(* IEC 61131-3 sources: std_i2980_v2.06_cp053/Source/IMM/ieccontrol/ODC1 (part 9) *)

END_TRANSITION
(* end sfc-code *)

END_ALGORITHM

(*
Run the auto cycle.
When the cycle has finished and mbStopCycle OR mbStopAfterCycle are true
opmode is automatically switched to manual and the PROCESS_ALGORITHM stops itself.
*)

PROCESS_ALGORITHM paRunAutomaticMovements ON TaskSequencer

#BEGIN_EDIT_BLOCK
(**************************************** WARNING ********************************************
 *** The KEBA Kemro K2 System including software is not intended for safety control tasks! ***
 ***                       For further information see Comment tab!                        ***
 *********************************************************************************************)

//call autoCycle
aRunAutoCycle(bStopCycle := mbStopCycle,
              bStopAfterCycle := mbStopAfterCycle);

IF aRunAutoCycle.bReady AND (mbStopCycle OR mbStopAfterCycle) THEN
   sv_bAutoCycleRunning := FALSE;
   // switch to manual mode and stop self at end of cycle
   fbAutoManual();

   abInterpreter.aResetStepMode();
   STOP_PROCESS_ALGORITHM(paCycleTime);
   STOP_PROCESS_ALGORITHM(paCycleTimeMachine);
   STOP_PROCESS_ALGORITHM();
END_IF;

;#END_EDIT_BLOCK END_ALGORITHM

(*
Cause initialisation of ODC sequence after startup(sv_bInitDone)
*)

POSTUPDATE_ALGORITHM pInitDone ON PU_Task_3 WITH sv_bInitDone

#BEGIN_EDIT_BLOCK
(**************************************** WARNING ********************************************
 *** The KEBA Kemro K2 System including software is not intended for safety control tasks! ***
 ***                       For further information see Comment tab!                        ***
 *********************************************************************************************)

fbDebugTrace2(nODCInterpreter,'Reloading ODC files because of sv_bInitDone');

IF sv_bUseProgramSwitches THEN
   //use program switches
   aSetPendingRecalc(RecalcMode := nODCRecalcReloadFiles);
ELSE
   //use existing sequence and only recalc internal arrays
   aSetPendingRecalc(RecalcMode := nODCRecalcInternal);
END_IF;

aDoPendingRecalc();
IF aDoPendingRecalc.bStartedRecalc THEN
   fbDebugTrace2(nDeviceState, 'recalc because pInitDone');
END_IF;

;#END_EDIT_BLOCK END_ALGORITHM

PROCESS_ALGORITHM paInit ON TaskMid AUTOSTART

VAR
 swoState : KSWO_Status;
END_VAR
#BEGIN_EDIT_BLOCK
(**************************************** WARNING ********************************************
 *** The KEBA Kemro K2 System including software is not intended for safety control tasks! ***
 ***                       For further information see Comment tab!                        ***
 *********************************************************************************************)

//initialize semaphore
Status := MovementsSema.Put();
IF Status <> KRTOS_Status_OK THEN
   dummy2 := ASSERT(FALSE, erAssert);
END_IF;

swoState := KSWO_AddVariable(Task := TaskInject,
                           Name := 'ActCycleTime',
                           Variable := sv_dCycleTime);

swoState := KSWO_AddVariable(Task := TaskAnalog,
                           Name := 'ActCycleTime',
                           Variable := sv_dCycleTime);

STOP_PROCESS_ALGORITHM();

;#END_EDIT_BLOCK END_ALGORITHM

(*
React to to operation mode changes and stop the autocycle immediately
when switching to setup/manual mode,
or reset cycle data when switching to Full/Halfauto operation mode.
*)

POSTUPDATE_ALGORITHM pOpmodeChanged ON PU_Task_7 WITH sv_OperationMode

#BEGIN_EDIT_BLOCK
(**************************************** WARNING ********************************************
 *** The KEBA Kemro K2 System including software is not intended for safety control tasks! ***
 ***                       For further information see Comment tab!                        ***
 *********************************************************************************************)

IF sv_OperationMode >= nHalfAutomatic THEN
   mbStopCycle := FALSE;
   mbStopAfterCycle := FALSE;
   (* back up sequence when machine is switched to auto mode
      and the sequence has changed *)
   START_PROCESS_ALGORITHM(paBackupSequence);

   (* PA stops itself again when finished *)
   START_PROCESS_ALGORITHM(paRunAutomaticMovements);
   START_PROCESS_ALGORITHM(paCycleTime);
   START_PROCESS_ALGORITHM(paCycleTimeMachine);
ELSIF sv_OperationMode < nHalfAutomatic THEN
   sv_bFirstCycle := TRUE;
   mbStopCycle := TRUE;
   mbCycleTimeRunning := FALSE;

   IF sv_StartedManualMovements.iStartedMovements = 0 THEN
      //recalc of sequence only if no movement is active
      //if there is still a movement active, the creation of a new sequence
      //will be triggered by postupdate algo pActiveMovements
      aDoPendingRecalc();
      IF aDoPendingRecalc.bStartedRecalc THEN
         fbDebugTrace2(nDeviceState, 'recalc because opmode change away from auto cycle');
      END_IF;
   END_IF;

END_IF;

;#END_EDIT_BLOCK END_ALGORITHM

(*
Handle evAlarmFinishCycleAndStop event which signals to stop after the end
of the current autocycle
*)

EVENT_ALGORITHM evaFinishCycleAndStop ON EV_Task_3 WITH evAlarmFinishCycleAndStop

VAR_INPUT
 evFinishCycleAndStopData : ALARM_EVENT_DATA;
END_VAR
#BEGIN_EDIT_BLOCK
(**************************************** WARNING ********************************************
 *** The KEBA Kemro K2 System including software is not intended for safety control tasks! ***
 ***                       For further information see Comment tab!                        ***
 *********************************************************************************************)

mbStopAfterCycle := TRUE;

;#END_EDIT_BLOCK END_ALGORITHM

POSTUPDATE_ALGORITHM pDataState ON PU_Task_3(1) WITH sv_DataState

VAR
 PrevState : tnDataState;
END_VAR
#BEGIN_EDIT_BLOCK
(**************************************** WARNING ********************************************
 *** The KEBA Kemro K2 System including software is not intended for safety control tasks! ***
 ***                       For further information see Comment tab!                        ***
 *********************************************************************************************)

IF sv_DataState = nReadMoldData THEN
   //loading of mold data in progress
   mbIgnoreProgramSwitchChange := TRUE;
   PrevState := nReadMoldData;
   sv_SequenceDimension.iMaxColumns := 0;
   sv_SequenceDimension.iMaxRows := 0;
ELSIF sv_DataState = nReadSequenceData THEN
   //loading of sequence in progress
   mbIgnoreProgramSwitchChange := TRUE;
   PrevState := nReadSequenceData;
   sv_SequenceDimension.iMaxColumns := 0;
   sv_SequenceDimension.iMaxRows := 0;
END_IF;

IF sv_DataState = nReady AND mbIgnoreProgramSwitchChange THEN

   //loading procedure ready
   mbIgnoreProgramSwitchChange := FALSE;

   //decide if only conditions should be recalculated (after loading sequence)
   //or complete sequence should be created (after program switch changed)
   IF sv_bUseProgramSwitches THEN
      aSetPendingRecalc(RecalcMode := nODCRecalcReloadFiles);
   ELSIF PrevState = nReadMoldData THEN
      aSetPendingRecalc(RecalcMode := nODCRecalcInternal);
   ELSIF PrevState = nReadSequenceData THEN
      aSetPendingRecalc(RecalcMode := nODCRecalcInternal);
   END_IF;

   aDoPendingRecalc();
   IF aDoPendingRecalc.bStartedRecalc THEN
      fbDebugTrace2(nDeviceState, 'recalc because data state change');
   END_IF;

   PrevState := nReady;
END_IF;

;#END_EDIT_BLOCK END_ALGORITHM

(*
React to program switch changes, and recalculate the ODC sequence.
*)

POSTUPDATE_ALGORITHM pDescriptionFilesChanged ON PU_Task_3 WITH sv_bODCFilesChanged

#BEGIN_EDIT_BLOCK
(**************************************** WARNING ********************************************
 *** The KEBA Kemro K2 System including software is not intended for safety control tasks! ***
 ***                       For further information see Comment tab!                        ***
 *********************************************************************************************)

IF NOT sv_bODCFilesChanged THEN
   RETURN;
END_IF;

sv_bODCFilesChanged := FALSE;

IF NOT sv_bInitDone THEN
   fbDebugTrace('ignoring sv_bODCFilesChanged because sv_bInitDone is FALSE');
   RETURN;
END_IF;

(* rebuild ODC array immediately with reloading files *)
aSetPendingRecalc(RecalcMode := nODCRecalcReloadFiles);

IF sv_OperationMode >= nHalfAutomatic THEN
   fbDebugTrace('skipping ODC recalc after file change because of OperationMode');
   RETURN;
END_IF;

IF sv_StartedMovements.iStartedMovements > 0 THEN
   fbDebugTrace('skipping ODC recalc after file change because there are started movements');
   RETURN;
END_IF;

aDoPendingRecalc();
IF aDoPendingRecalc.bStartedRecalc THEN
   fbDebugTrace2(nDeviceState, 'recalc because files changed');
END_IF;

;#END_EDIT_BLOCK END_ALGORITHM

(*
create internal array and calculate safety conditions after
teachmode becomes inactive
*)

POSTUPDATE_ALGORITHM pNewSequenceFromEditor ON PU_Task_3 WITH sv_iActiveEditors

VAR
 fbLockUnlock : FBLockUnlock := (DeviceId:=(CompId:=cCompOperationMode,IndexId:=1),MoveDir:=cModeAutomatic,MoveId:=cModeAutomatic);
END_VAR
#BEGIN_EDIT_BLOCK
(**************************************** WARNING ********************************************
 *** The KEBA Kemro K2 System including software is not intended for safety control tasks! ***
 ***                       For further information see Comment tab!                        ***
 *********************************************************************************************)

IF sv_iActiveEditors <> 0 THEN
   //teach mode active
   //avoid changing operation mode to HA or FA
   fbLockUnlock.Alarm.AlarmId := erTeachModeActive;
   fbLockUnlock.Mode := nLockAbort;
   fbLockUnlock();

   //reset sv_bUseProgramSwitches immediately after activating teach mode
   //so that "controlled by machine sequencer" is displayed instead of program switches
   sv_bUseProgramSwitches := FALSE;
   RETURN;
ELSE
   fbLockUnlock.Alarm.AlarmId := erTeachModeActive;
   fbLockUnlock.Mode := nUnlock;
   fbLockUnlock();
END_IF;

//teach mode inactive => new sequence programmed by editor
// -> create internal array, calculate safety conditions, do plaus checks
aSetPendingRecalc(RecalcMode := nODCRecalcInternal);

aDoPendingRecalc();
IF aDoPendingRecalc.bStartedRecalc THEN
   fbDebugTrace2(nDeviceState, 'recalc because new sequence from editor');
END_IF;

;#END_EDIT_BLOCK END_ALGORITHM

POSTUPDATE_ALGORITHM aRestoreSequenceBackup ON EV_Task_7 WITH sv_iSequenceToRestore

#BEGIN_EDIT_BLOCK
(**************************************** WARNING ********************************************
 *** The KEBA Kemro K2 System including software is not intended for safety control tasks! ***
 ***                       For further information see Comment tab!                        ***
 *********************************************************************************************)

IF sv_iSequenceToRestore = 0 THEN
   RETURN;
END_IF;

IF sv_iSequenceToRestore > cODCSequenceBackupCount THEN
   fbDebugTrace2(nODCInterpreter, 'restoring actual sequence calculated from switches');
   aSetPendingRecalc(RecalcMode := nODCRecalcCylce);
END_IF;

fbDebugTrace2(nODCInterpreter, CONCAT('restoring old sequence ', DINT_TO_STRING(sv_iSequenceToRestore)));
sv_ODCSequence := sv_ODCSequenceBackup[sv_iSequenceToRestore].Sequence;
aSetPendingRecalc(RecalcMode := nODCRecalcSafety);
aDoPendingRecalc(); //FIXME: this may not do more than security recalculation -> otherwise loaded array would be overwritten
IF aDoPendingRecalc.bStartedRecalc THEN
   fbDebugTrace2(nDeviceState, 'recalc because sequence backup is restored');
END_IF;
sv_iSequenceToRestore := 0;
fbDebugTrace2(nODCInterpreter, 'restoring old sequence done');

;#END_EDIT_BLOCK END_ALGORITHM

(*
React to program switch changes, and recalculate the ODC sequence.
*)

POSTUPDATE_ALGORITHM pProgramSwitchChanged ON PU_Task_3 WITH sv_bProgramSwitchChanged

#BEGIN_EDIT_BLOCK
(**************************************** WARNING ********************************************
 *** The KEBA Kemro K2 System including software is not intended for safety control tasks! ***
 ***                       For further information see Comment tab!                        ***
 *********************************************************************************************)

IF NOT sv_bProgramSwitchChanged THEN
   RETURN;
END_IF;

sv_bProgramSwitchChanged := FALSE;

IF NOT sv_bInitDone THEN
   fbDebugTrace2(nODCInterpreter, 'ignoring program switch change because sv_bInitDone is FALSE');
   RETURN;
END_IF;

IF NOT sv_bUseProgramSwitches THEN
   // ignore changing of program switch if sequence from graphical editor is used
   fbDebugTrace2(nODCInterpreter, 'ignoring program switch change because of sv_bUseProgramSwitches');
   RETURN;
END_IF;

IF mbIgnoreProgramSwitchChange THEN
   fbDebugTrace2(nODCInterpreter, 'ignoring program switch change because of sv_DataState');
   RETURN;
END_IF;

aSetPendingRecalc(RecalcMode := nODCRecalcCylce);

IF sv_OperationMode >= nHalfAutomatic THEN
   fbDebugTrace('skipping ODC recalc after program switch change because of OperationMode');
   RETURN;
END_IF;

IF sv_StartedMovements.iStartedMovements > 0 THEN
   fbDebugTrace('skipping ODC recalc after program switch change because there are started movements');
   RETURN;
END_IF;

(* rebuild ODC array immediately without reloading files *)
aDoPendingRecalc();
IF aDoPendingRecalc.bStartedRecalc THEN
   fbDebugTrace2(nDeviceState, 'recalc because program switch changed');
END_IF;

;#END_EDIT_BLOCK END_ALGORITHM

(*
React to program switch changes, and recalculate the ODC sequence.
*)

POSTUPDATE_ALGORITHM pActivationChanged ON PU_Task_3 WITH sv_bActivationChanged

#BEGIN_EDIT_BLOCK
(**************************************** WARNING ********************************************
 *** The KEBA Kemro K2 System including software is not intended for safety control tasks! ***
 ***                       For further information see Comment tab!                        ***
 *********************************************************************************************)

IF NOT sv_bActivationChanged THEN
   RETURN;
END_IF;

sv_bActivationChanged := FALSE;

IF NOT sv_bInitDone THEN
   fbDebugTrace('ignoring sv_bActivationChanged because sv_bInitDone is FALSE');
   RETURN;
END_IF;

IF mbIgnoreProgramSwitchChange THEN
   fbDebugTrace2(nODCInterpreter, 'ignoring activation change because of sv_DataState');
   RETURN;
END_IF;

(* recalculate ODC safety without reloading files/recalculating the sequence *)
aSetPendingRecalc(RecalcMode := nODCRecalcSafety);

IF sv_OperationMode >= nHalfAutomatic THEN
   fbDebugTrace('skipping ODC recalc after activation change because of OperationMode');
   RETURN;
END_IF;

IF sv_StartedMovements.iStartedMovements > 0 THEN
   fbDebugTrace('skipping ODC recalc after activation change because there are started movements');
   RETURN;
END_IF;

aDoPendingRecalc();
IF aDoPendingRecalc.bStartedRecalc THEN
   fbDebugTrace2(nDeviceState, 'recalc because activation change');
END_IF;

;#END_EDIT_BLOCK END_ALGORITHM

PROCESS_ALGORITHM paVersionInfo ON TaskSlow AUTOSTART

VAR
 b : BOOL;
END_VAR
#BEGIN_EDIT_BLOCK
(**************************************** WARNING ********************************************
 *** The KEBA Kemro K2 System including software is not intended for safety control tasks! ***
 ***                       For further information see Comment tab!                        ***
 *********************************************************************************************)

b := FCreateODCVersion();
STOP_PROCESS_ALGORITHM();

;#END_EDIT_BLOCK END_ALGORITHM

(*
trigger creation of sequence by program switches
*)

POSTUPDATE_ALGORITHM pChangeToProgramSwitches ON PU_Task_7 WITH sv_bUseProgramSwitches

VAR_TEMP
 iDevice : DINT;
END_VAR
#BEGIN_EDIT_BLOCK
(**************************************** WARNING ********************************************
 *** The KEBA Kemro K2 System including software is not intended for safety control tasks! ***
 ***                       For further information see Comment tab!                        ***
 *********************************************************************************************)

IF mbIgnoreProgramSwitchChange THEN
   //loading procedure in progress
   RETURN;
END_IF;

IF sv_bUseProgramSwitches THEN
   //activate all devices after a change from
   //machine sequencer mode to program switch mode
   FOR iDevice := 1 TO sv_ODCDeviceMovements.iCount DO
      IF CHECK_REF(sv_ODCDeviceMovements.Devices[iDevice].pbDeviceActivated^) THEN
         sv_ODCDeviceMovements.Devices[iDevice].pbDeviceActivated^ := TRUE;
      END_IF;
   END_FOR;

   //create new sequence depending on the program switches
   //set mode to nODCRecalcReloadFiles because maybe sequence was
   //never created with program switches before
   aSetPendingRecalc(RecalcMode := nODCRecalcReloadFiles);
   aDoPendingRecalc();
   IF aDoPendingRecalc.bStartedRecalc THEN
      fbDebugTrace2(nDeviceState, 'recalc because change to program switch mode');
   END_IF;
END_IF;

;#END_EDIT_BLOCK END_ALGORITHM

(*
This algorithm checks the start conditions for the cycle if the
operator switches to half or fullauto cycle.
Safety relevant devices must be in the position which they should have according
the programmed cycle.
Not safety relevant devices must be in their default position.
Deactivated devices and devices which have no default position are not checked.
*)

ALGORITHM aCheckCycleStartConditions

VAR_TEMP
 iDevice : DINT;
END_VAR

VAR
 Pos : tsODCStepPos;
 DeviceId : tsDeviceId;
 SafetyArray : tyODCDependencyArray;
 iDefaultMove : DINT;
 bAllowed : BOOL;
 abODCCheckDependencies : ABODCCheckDependencies;
 fbCheckPosReached : FBCheckPosReached;
 bEjectorIgnored : BOOL;
 EjectorDependency : LWORD;
END_VAR
#BEGIN_EDIT_BLOCK
(**************************************** WARNING ********************************************
 *** The KEBA Kemro K2 System including software is not intended for safety control tasks! ***
 ***                       For further information see Comment tab!                        ***
 *********************************************************************************************)

Pos.iColumn := 1;
Pos.iRow := 1;

DeviceId.CompId := sv_ODCSequence[1,1].iCompId;
DeviceId.IndexId := INT_TO_DINT(sv_ODCSequence[1,1].iIndexId);

//check safety array of first step (ODC.BeginSequence)
bEjectorIgnored := FALSE;
IF mbEjeBwdAtCycleStart THEN
   //ejector must not be bwd when operator switches to HA or FA
   //the ejector bwd movement is done in aRunAutoCylce
   //=> start of cycle should be possible if ejector is not bwd)
   //=> dependency must be modified for this case
   //all other safety relevant movements (mold, cores, ...) must be in the calculated startposition
   EjectorDependency := sv_ODCSequenceInt[1,1].SafetyArray[miIndexEjectorInSafetyArray].Dependency;
   sv_ODCSequenceInt[1,1].SafetyArray[miIndexEjectorInSafetyArray].Dependency := cNoDependency;
   bEjectorIgnored := TRUE;
END_IF;

//check init safety array
//(check all safety relevant devices)
abODCCheckDependencies.aCheck(StepPos := Pos, DeviceIdSelf := DeviceId);
bAllowed := abODCCheckDependencies.aCheck.bAllowed;

//write back the original value
IF bEjectorIgnored THEN
   sv_ODCSequenceInt[1,1].SafetyArray[miIndexEjectorInSafetyArray].Dependency := EjectorDependency;
END_IF;

//check state of not safety relevant devices
//always check even if safety relevant check already failed
SafetyArray := sv_ODCSequenceInt[1,1].SafetyArray;
FOR iDevice := 1 TO sv_ODCDeviceMovements.iCount DO
   DeviceId := sv_ODCDeviceMovements.Devices[iDevice].DeviceId;
   iDefaultMove := sv_ODCDeviceMovements.Devices[iDevice].iDefaultMoveNumber;

   IF (SafetyArray[iDevice].Dependency = cNoDependency) AND (DeviceId.CompId <> cCompODC) THEN
      //device not safety relevant
      IF sv_ODCDeviceMovements.Devices[iDevice].pbDeviceActivated^ AND iDefaultMove <> 0 THEN
         //if device is activated and a default movement is available,
         //the default movement of this device must be in endposition
         fbCheckPosReached(DeviceId := DeviceId,
                           MoveDir := sv_MovementsAvailable[iDefaultMove].pMovementData^.MoveDir,
                           MoveId := sv_MovementsAvailable[iDefaultMove].pMovementData^.MoveId);

         IF NOT fbCheckPosReached.bPosReached THEN
            IF sv_TraceLevel.bODCInterpreter THEN
               fbDebugTrace(CONCAT('cycle start not allowed by default position check of ',
                                   DINT_TO_STRING(DeviceId.CompId), '.', DINT_TO_STRING(DeviceId.IndexId),
                                   ' -> setting alarm ',
                                   GET_ALARM_NAME(fbCheckPosReached.Alarm.AlarmId)));
            END_IF;
            //set according alarm
            SET_ALARM(Name := fbCheckPosReached.Alarm.AlarmId,
                      SubID1 := fbCheckPosReached.Alarm.SubId[1],
                      SubID2 := fbCheckPosReached.Alarm.SubId[2],
                      SubID3 := fbCheckPosReached.Alarm.SubId[3],
                      SubID4 := fbCheckPosReached.Alarm.SubId[4]);
            bAllowed := FALSE;
         END_IF;
      END_IF;
   END_IF;
END_FOR;

IF NOT bAllowed THEN
   IF sv_TraceLevel.bODCInterpreter THEN
      fbDebugTrace('checking cycle start conditions found problems -> switching back to manual mode');
   END_IF;
   //switch away from auto mode if any check fails
   fbAutoManual();
END_IF;

;#END_EDIT_BLOCK END_ALGORITHM

POSTUPDATE_ALGORITHM pOperationMode ON PU_Task_7 WITH sv_OperationMode

VAR_TEMP
 sOperationMode : STRING(255);
END_VAR

VAR
 PrevOpMode : tnOperationMode := nManual;
END_VAR
#BEGIN_EDIT_BLOCK
(**************************************** WARNING ********************************************
 *** The KEBA Kemro K2 System including software is not intended for safety control tasks! ***
 ***                       For further information see Comment tab!                        ***
 *********************************************************************************************)

IF sv_TraceLevel.bODCInterpreter THEN
   //trace opmode switch
   IF sv_OperationMode = nSetup THEN
      sOperationMode := 'Setup';
   ELSIF sv_OperationMode = nManual THEN
      sOperationMode := 'Manual';
   ELSIF sv_OperationMode = nHalfAutomatic THEN
      sOperationMode := 'HalfAutomatic';
   ELSIF sv_OperationMode = nFullAutomatic THEN
      sOperationMode := 'FullAutomatic';
   ELSE
      sOperationMode := '???';
   END_IF;
   fbDebugTrace(CONCAT('sv_OperationMode changed to ', sOperationMode));
END_IF;

IF PrevOpMode < nHalfAutomatic AND sv_OperationMode >= nHalfAutomatic THEN
   //check cycle start conditions
   aCheckCycleStartConditions();
END_IF;

PrevOpMode := sv_OperationMode;

;#END_EDIT_BLOCK END_ALGORITHM

PROCESS_ALGORITHM paRunManualCombinedMovement ON TaskSequencer

(* IecGraph-Code *)

(* init step *)
INITIAL_STEP SInit:
END_STEP

(* steps *)
STEP S_Run:
Action24 (P);
ARunCombinedMovement (N);
END_STEP

ACTION Action24: #BEGIN_EDIT_BLOCK
sv_bODCCombinedMoveActive := TRUE;

;#END_EDIT_BLOCK END_ACTION (*Action24*)
ACTION ARunCombinedMovement: #BEGIN_EDIT_BLOCK
// run a combined movements
abInterpreter.aInterpret();
abInterpreter.aStatus();

;#END_EDIT_BLOCK END_ACTION (*ARunCombinedMovement*)
STEP S_Finished:
ATrace (P);
END_STEP

STEP S_StopInterpreter:
AStopInterpreter (P);
END_STEP

ACTION AStopInterpreter: #BEGIN_EDIT_BLOCK
abInterpreter.aStopInterpreterNormal();

;#END_EDIT_BLOCK END_ACTION (*AStopInterpreter*)
STEP S_NotActive:
ATraceNotActive (P);
END_STEP

STEP S_Error:
ATraceError (P);
END_STEP

STEP S_Recalc:
ADoPendingRecalc (P);
END_STEP

STEP S_Stop:
AStop (P);
END_STEP

ACTION AStop: #BEGIN_EDIT_BLOCK
sv_bODCCombinedMoveActive := FALSE;
STOP_PROCESS_ALGORITHM();

;#END_EDIT_BLOCK END_ACTION (*AStop*)

(* transitions *)
GO_ON_TRANSITION Trans1 (* Trans1 *) FROM SInit TO S_Run :=  #BEGIN_EDIT_BLOCK
TRUE
;#END_EDIT_BLOCK
END_TRANSITION

GO_ON_TRANSITION TFinished (* Trans2 *) FROM S_Run TO S_Finished :=  #BEGIN_EDIT_BLOCK
abInterpreter.aStatus.bFinished
;#END_EDIT_BLOCK
END_TRANSITION

GO_ON_TRANSITION TAllMovementsReady (* Trans7 *) FROM S_Finished TO S_StopInterpreter :=  #BEGIN_EDIT_BLOCK
sv_StartedManualMovements.iStartedMovements = 0
;#END_EDIT_BLOCK
(*Interpreter is finished -> wait untill all movements
are ready  (for example airvalve can still be active)*)
END_TRANSITION

GO_ON_TRANSITION Trans11 (* Trans11 *) FROM S_StopInterpreter TO S_Recalc :=  #BEGIN_EDIT_BLOCK
TRUE
;#END_EDIT_BLOCK
END_TRANSITION

GO_ON_TRANSITION TNotActive (* Trans5 *) FROM S_Run TO S_NotActive :=  #BEGIN_EDIT_BLOCK
NOT abInterpreter.aStatus.bActive
;#END_EDIT_BLOCK
END_TRANSITION

GO_ON_TRANSITION Trans8 (* Trans8 *) FROM S_NotActive TO S_Recalc :=  #BEGIN_EDIT_BLOCK
TRUE
;#END_EDIT_BLOCK
END_TRANSITION

GO_ON_TRANSITION TError (* Trans6 *) FROM S_Run TO S_Error :=  #BEGIN_EDIT_BLOCK
abInterpreter.aStatus.bError
;#END_EDIT_BLOCK
END_TRANSITION

GO_ON_TRANSITION Trans9 (* Trans9 *) FROM S_Error TO S_Recalc :=  #BEGIN_EDIT_BLOCK
TRUE
;#END_EDIT_BLOCK
END_TRANSITION

GO_ON_TRANSITION Trans12 (* Trans12 *) FROM S_Recalc TO S_Stop :=  #BEGIN_EDIT_BLOCK
TRUE
;#END_EDIT_BLOCK
END_TRANSITION

TRANSITION Trans4 (* Trans4 *) FROM S_Stop TO S_Run :=  #BEGIN_EDIT_BLOCK
TRUE
;#END_EDIT_BLOCK
END_TRANSITION

(* end IecGraph-Code *)
(* sfc-code *)

(* stand alone actions *)
ACTION ATrace: #BEGIN_EDIT_BLOCK
(**************************************** WARNING ********************************************
 *** The KEBA Kemro K2 System including software is not intended for safety control tasks! ***
 ***                       For further information see Comment tab!                        ***
 *********************************************************************************************)

fbDebugTrace2(nODCInterpreter,'stopping combined movement PA because interpreter has finished');
IF sv_StartedManualMovements.iStartedMovements <> 0 THEN
   fbDebugTrace2(nODCInterpreter,'There were still some movements active at end of a combined movement');
END_IF;

;#END_EDIT_BLOCK END_ACTION (*ATrace*)
ACTION ATraceError: #BEGIN_EDIT_BLOCK
(**************************************** WARNING ********************************************
 *** The KEBA Kemro K2 System including software is not intended for safety control tasks! ***
 ***                       For further information see Comment tab!                        ***
 *********************************************************************************************)

fbDebugTrace2(nODCInterpreter,'stopping combined movement PA because interpreter reported an error');

;#END_EDIT_BLOCK END_ACTION (*ATraceError*)
ACTION ATraceNotActive: #BEGIN_EDIT_BLOCK
(**************************************** WARNING ********************************************
 *** The KEBA Kemro K2 System including software is not intended for safety control tasks! ***
 ***                       For further information see Comment tab!                        ***
 *********************************************************************************************)

fbDebugTrace2(nODCInterpreter,'stopping combined movement PA because interpreter is not active anymore');
IF sv_StartedManualMovements.iStartedMovements <> 0 THEN
   fbDebugTrace2(nODCInterpreter,'There were still some movements active at end of a combined movement');
END_IF;

;#END_EDIT_BLOCK END_ACTION (*ATraceNotActive*)
ACTION ADoPendingRecalc: #BEGIN_EDIT_BLOCK
(**************************************** WARNING ********************************************
 *** The KEBA Kemro K2 System including software is not intended for safety control tasks! ***
 ***                       For further information see Comment tab!                        ***
 *********************************************************************************************)

IF sv_StartedManualMovements.iStartedMovements = 0 THEN
   //all movements ready
   aDoPendingRecalc();
   IF aDoPendingRecalc.bStartedRecalc THEN
      fbDebugTrace2(nDeviceState, 'recalc because interpreter finished and iStartedMovements = 0');
   END_IF;
END_IF;

;#END_EDIT_BLOCK END_ACTION (*ADoPendingRecalc*)
(* end sfc-code *)

END_ALGORITHM

(*
supervision of check conditions for single movements in
manual and setup mode
For combined movements and in half and fullauto cycle the supervision
is done by the interpreter
*)

PROCESS_ALGORITHM paCheckConditionsManual ON TaskAnalog

VAR_TEMP
 i : DINT;
END_VAR

VAR
 TmpStepPos : tsODCStepPos;
END_VAR
#BEGIN_EDIT_BLOCK
(**************************************** WARNING ********************************************
 *** The KEBA Kemro K2 System including software is not intended for safety control tasks! ***
 ***                       For further information see Comment tab!                        ***
 *********************************************************************************************)

FOR i := 1 TO sv_StartedManualMovements.iStartedMovements DO

   TmpStepPos := sv_StartedManualMovements.MoveData[i].StepPos;
   IF (TmpStepPos.iColumn <> 0) AND (TmpStepPos.iRow <> 0) THEN
      //if a combined movement (sequence) is active, the supervision of the check conditions
      //is done automatically by the interpreter
      abInterpreter.aCheckConditionsManual(Movement := sv_ODCSequence[TmpStepPos.iColumn][TmpStepPos.iRow], bNoAlarms := FALSE);

      IF NOT abInterpreter.aCheckConditionsManual.bCheckConditionsOk THEN
         //check condition not ok
         abInterpreter.aStopInterpreterError();
      END_IF;
   END_IF;
END_FOR;

;#END_EDIT_BLOCK END_ALGORITHM

PROCESS_ALGORITHM paCycleTime ON TaskInject

VAR
 b : BOOL;
 fbTonCycleTime : TON;
END_VAR
#BEGIN_EDIT_BLOCK
(**************************************** WARNING ********************************************
 *** The KEBA Kemro K2 System including software is not intended for safety control tasks! ***
 ***                       For further information see Comment tab!                        ***
 *********************************************************************************************)

//Cycle time - from start to start
IF mbCycleTimeRunning THEN

   IF mbResetCycleTime THEN
      fbTonCycleTime(IN := FALSE);
      mbResetCycleTime := FALSE;
   END_IF;

   fbTonCycleTime(IN := TRUE,
                  PT := t#20d);

   b := WRITE_SV_DIRECT(sv_dCycleTime, fbTonCycleTime.ET);

   IF sv_dCycleTime > sv_dMaxCycleTime THEN
      SET_ALARM(Name := erCycleTimeExceeded);
   END_IF;
END_IF;

;#END_EDIT_BLOCK END_ALGORITHM

PROCESS_ALGORITHM paCycleTimeMachine ON TaskMid

VAR
 b : BOOL;
 fbTonCycleTimeMachine : TON (* Clock the cycletime from start to end of cycle *);
END_VAR
#BEGIN_EDIT_BLOCK
(**************************************** WARNING ********************************************
 *** The KEBA Kemro K2 System including software is not intended for safety control tasks! ***
 ***                       For further information see Comment tab!                        ***
 *********************************************************************************************)

//Cycle time machine - from start to end of cycle
IF mbCycleTimeRunning AND mbCycleTimeMachineRunning THEN

   IF mbResetCycleTimeMachine THEN
      fbTonCycleTimeMachine(IN := FALSE);
      mbResetCycleTimeMachine := FALSE;
   END_IF;

   fbTonCycleTimeMachine(IN := TRUE,
                         PT := t#20d);

   b := WRITE_SV_DIRECT(sv_dCycleTimeMachine, fbTonCycleTimeMachine.ET);
END_IF;

;#END_EDIT_BLOCK END_ALGORITHM

POSTUPDATE_ALGORITHM pSequenceInterruption ON PU_Task_13 WITH sv_bSequenceInterruption

VAR
 dummy : DINT;
END_VAR
#BEGIN_EDIT_BLOCK
(**************************************** WARNING ********************************************
 *** The KEBA Kemro K2 System including software is not intended for safety control tasks! ***
 ***                       For further information see Comment tab!                        ***
 *********************************************************************************************)

IF sv_bSequenceInterruption THEN
   IF sv_TraceLevel.bODCInterpreter THEN
      dummy := Print('***** INTERRUPT SEQUENCE *****');
   END_IF;
   mbStopAfterCycle := TRUE;
   abInterpreter.aInterruptSequence();
ELSE
   sv_bStepBwdActive := FALSE;
   IF sv_OperationMode >= nHalfAutomatic THEN
      IF sv_TraceLevel.bODCInterpreter THEN
         dummy := Print('***** CONTINUE SEQUENCE *****');
      END_IF;
      abInterpreter.aContinueSequence();
      mbStopAfterCycle := FALSE;
   END_IF;
END_IF;

;#END_EDIT_BLOCK END_ALGORITHM

ALGORITHM aStartInverseMovement

VAR_INPUT
 iMoveNr : DINT;
 iColumn : DINT;
END_VAR

VAR_TEMP
 i : DINT;
END_VAR

VAR
 iFuIndex : DINT;
 iMoveIdInverse : tMoveIdent;
END_VAR
#BEGIN_EDIT_BLOCK
(**************************************** WARNING ********************************************
 *** The KEBA Kemro K2 System including software is not intended for safety control tasks! ***
 ***                       For further information see Comment tab!                        ***
 *********************************************************************************************)

//get inverse movement
iMoveIdInverse := sv_MovementsAvailable[iMoveNr].pMovementData^.iMoveIdInverseMovement;
IF iMoveIdInverse = cMinMoveIdent THEN
   //no inverse movement defined
   //set alarm if moenet does not belong to ODC - function unit
   IF (sv_MovementsAvailable[iMoveNr].DeviceId <> sv_DeviceId) THEN
      SET_ALARM(Name := erNoInverseMovement,
                SubID1 := sv_MovementsAvailable[iMoveNr].DeviceId.CompId,
                SubID2 := sv_MovementsAvailable[iMoveNr].DeviceId.IndexId,
                SubID3 := sv_MovementsAvailable[iMoveNr].pMovementData^.MoveId);
   END_IF;

   RETURN; //return here
END_IF;

iFuIndex := sv_MovementsAvailable[iMoveNr].iFuIndex;
FOR i := 1 TO sv_ODCDeviceMovements.Devices[iFuIndex].iNumberOfMovements DO
   IF sv_ODCDeviceMovements.Devices[iFuIndex].Movements[i]^.MoveId = iMoveIdInverse THEN
      //inverse movement found => try to start it
      aStartSingleMovement(DeviceId := sv_ODCDeviceMovements.Devices[iFuIndex].DeviceId,
                           MoveDir := sv_ODCDeviceMovements.Devices[iFuIndex].Movements[i]^.MoveDir,
                           MoveId := sv_ODCDeviceMovements.Devices[iFuIndex].Movements[i]^.MoveId,
                           IntermediateCond := 0,
                           bNeedCheckSafety := (sv_ODCDeviceMovements.Devices[iFuIndex].Movements[i]^.iSafetyIdentifier > 0));

      IF aStartSingleMovement.bStarted THEN
         mActiveStepBwdMovements[iColumn].DeviceId := sv_ODCDeviceMovements.Devices[iFuIndex].DeviceId;
         mActiveStepBwdMovements[iColumn].MoveId := sv_ODCDeviceMovements.Devices[iFuIndex].Movements[i]^.MoveId;
         mActiveStepBwdMovements[iColumn].MoveDir := sv_ODCDeviceMovements.Devices[iFuIndex].Movements[i]^.MoveDir;
      END_IF;

      EXIT;
   END_IF;
END_FOR;

;#END_EDIT_BLOCK END_ALGORITHM

POSTUPDATE_ALGORITHM pStepFwd ON PU_Task_3 WITH di_StepFwd

#BEGIN_EDIT_BLOCK
(**************************************** WARNING ********************************************
 *** The KEBA Kemro K2 System including software is not intended for safety control tasks! ***
 ***                       For further information see Comment tab!                        ***
 *********************************************************************************************)

IF NOT sv_bSequenceInterruption THEN
   //button is only working if sequence is interrupted
   RETURN;
END_IF;

IF di_StepFwd THEN
   //trigger interpreter to execute the next step(s)
   IF sv_StartedManualMovements.iStartedMovements = 0 THEN
      //ignore step fwd button if any movment is active
      abInterpreter.aEnableNextStep();
   END_IF;
ELSE
   //stop actually executed step(s)
   abInterpreter.aInterruptSequence();
END_IF;

;#END_EDIT_BLOCK END_ALGORITHM

POSTUPDATE_ALGORITHM pStepBwd ON PU_Task_3 WITH di_StepBwd

VAR_TEMP
 iColumn : DINT;
END_VAR

VAR
 iActiveMoveNr : DINT;
END_VAR
#BEGIN_EDIT_BLOCK
(**************************************** WARNING ********************************************
 *** The KEBA Kemro K2 System including software is not intended for safety control tasks! ***
 ***                       For further information see Comment tab!                        ***
 *********************************************************************************************)

IF NOT sv_bSequenceInterruption THEN
   //button is only working if sequence is interrupted
   RETURN;
END_IF;

IF di_StepBwd THEN

   IF sv_StartedManualMovements.iStartedMovements <> 0 THEN
      //ignore step bwd button if any movement is still active
      RETURN;
   END_IF;

   sv_bStepBwdActive := TRUE;

   //get actual active lines and find the inverse movements
   FOR iColumn := 1 TO sv_iUsedColumns DO
      IF sv_InterpreterParallelInfo[iColumn].bColumnActive THEN
         //it is possible that the sequence was interrupted during waiting
         //for completion of a parallel tree -> in this case the line number must be decreased
         IF (sv_ODCSequence[iColumn, sv_InterpreterParallelInfo[iColumn].iRow].iMoveId = cMoveEndParallel) THEN
            abInterpreter.aDecreaseRow(bStartInActualLine := FALSE,
                                       iColumn := iColumn,
                                       iEndRow := 1);
         ELSIF (sv_ODCSequence[iColumn, sv_InterpreterParallelInfo[iColumn].iRow].iMoveId = cMoveStartParallel) OR
            (sv_ODCSequence[iColumn, sv_InterpreterParallelInfo[iColumn].iRow].iMoveId = cMoveStartParallelOpen) THEN
            //stepping bwd stopped during waiting for parallel trees
            //-> check actual state of this tree
            abInterpreter.aDecreaseRow(bStartInActualLine := TRUE,
                                       iColumn := iColumn,
                                       iEndRow := 1);
         END_IF;

         iActiveMoveNr := sv_ODCSequenceInt[iColumn, sv_InterpreterParallelInfo[iColumn].iRow].iMoveNumber;
         IF iActiveMoveNr > cMoveNone THEN
            aStartInverseMovement(iMoveNr := iActiveMoveNr,
                                 iColumn := iColumn);
         END_IF;
      END_IF;
   END_FOR;
ELSE
   //stop actually executed step(s)
   abInterpreter.aInterruptSequence();

   sv_bStepBwdActive := FALSE;
END_IF;

;#END_EDIT_BLOCK END_ALGORITHM

EVENT_ALGORITHM evaModifyCycleStartCondition ON EV_Task_3 WITH evModifyCycleStartCondition

VAR_INPUT
 evModifyCycleStartCondData : tevModifyCycleStartCondData;
END_VAR

VAR_TEMP
 i : DINT;
END_VAR

VAR
 dummy : DINT;
 eventData : tevModifyCycleStartCondData;
 iFuIndex : DINT;
 iMoveNr : DINT;
 fbAddDependency : FBAddDependency;
 fbGetMoveNumber : FBGetMoveNumber;
END_VAR
#BEGIN_EDIT_BLOCK
(**************************************** WARNING ********************************************
 *** The KEBA Kemro K2 System including software is not intended for safety control tasks! ***
 ***                       For further information see Comment tab!                        ***
 *********************************************************************************************)

IF sv_iInitOK <> 20 THEN
   dummy := Print('!!! evModifyCycleStartCondition event ignored !!!');
   RETURN; //ignore event because machine sequence is not created
END_IF;

//save event data
eventData := evModifyCycleStartCondData;

//get index of this device in the safety array
iFuIndex := 0;
FOR i := 1 TO sv_ODCDeviceMovements.iCount DO
   IF sv_ODCDeviceMovements.Devices[i].DeviceId = eventData.DeviceId THEN
      iFuIndex := i;
      EXIT;
   END_IF;
END_FOR;

IF iFuIndex = 0 THEN
   RETURN; //device not found
END_IF;

IF (eventData.iMode = 1) THEN
   //get movement number
   fbGetMoveNumber(DeviceId := eventData.DeviceId,
                  MoveId := eventData.MoveId,
                  MoveDir := eventData.MoveDir);

   IF fbGetMoveNumber.bFound THEN
      iMoveNr := fbGetMoveNumber.iMoveNumber;
   ELSE
      RETURN; //movement not found
   END_IF;

   //add this movement as additional start condition of this device
   fbAddDependency(iFuIndex := iFuIndex,
                   iMoveNr := iMoveNr,
                   iCount := eventData.iCount,
                   iMode := 1,
                   Dependency := sv_ODCSequenceInt[1,1].SafetyArray);

ELSE
   ; //unsupported mode
END_IF;

;#END_EDIT_BLOCK END_ALGORITHM

END_ALGORITHM_BLOCK

#END_OF_IEC_PART

@Puma @IecEditor 6 97 @Pou 25
@@@BEG_Comment@@@
@h    ! WARNING !
@h    The Kemro K2 system (including software) only meets category B according to EN 954-1,
@h    thus it is not intended for usage in safety-relevant control applications in the field
@h    of personal safety (e.g. emergency stop).
@h    To implement potentially necessary safety-relevant control tasks, always use additional
@h    external safety devices that are intended for the particular purpose, and meet the necessary
@h    functional safety.
@h    For further information see EN 954-1 (EN ISO 13849-1) and/or the K2-x00 user manual, chapter
@h    "CE conformity, directives and standards".

@@@END_Comment@@@

@BEG_Contents

@BEG_Func
@RT(17)FuncTreeContainer
7
@Var @RT(9)SET_ALARM @RT(0) @T @T @DERIVED 0 @F @RT(23)KEBA_STANDARD_PROCEDURE @F
@T
@BEG_Attrib
0 @RT(0) @RT(0)
@END_Attrib
1 1 @F @F @F @F

@Var @RT(23)START_PROCESS_ALGORITHM @RT(0) @T @T @DERIVED 0 @F @RT(23)KEBA_STANDARD_PROCEDURE @F
@T
@BEG_Attrib
0 @RT(0) @RT(0)
@END_Attrib
1 1 @F @F @F @F

@Var @RT(9)CHECK_REF @RT(0) @T @T @DERIVED 0 @F @RT(23)KEBA_STANDARD_PROCEDURE @F
@T
@BEG_Attrib
0 @RT(0) @RT(0)
@END_Attrib
1 1 @F @F @F @F

@Var @RT(22)STOP_PROCESS_ALGORITHM @RT(0) @T @T @DERIVED 0 @F @RT(23)KEBA_STANDARD_PROCEDURE @F
@T
@BEG_Attrib
0 @RT(0) @RT(0)
@END_Attrib
1 1 @F @F @F @F

@Var @RT(17)FCreateODCVersion @RT(0) @T @T @DERIVED 0 @F @RT(8)FUNCTION @F
@T
@BEG_Attrib
0 @RT(0) @RT(0)
@END_Attrib
1 1 @F @F @F @F

@Var @RT(9)SET_EVENT @RT(0) @T @T @DERIVED 0 @F @RT(23)KEBA_STANDARD_PROCEDURE @F
@T
@BEG_Attrib
0 @RT(0) @RT(0)
@END_Attrib
1 1 @F @F @F @F

@Var @RT(24)FGetCatConfigValueString @RT(0) @T @T @DERIVED 0 @F @RT(8)FUNCTION @F
@T
@BEG_Attrib
0 @RT(0) @RT(0)
@END_Attrib
1 1 @F @F @F @F

@END_Func

@BEG_Const
@RT(18)ConstTreeContainer
30
@Var @RT(13)cMinMoveIdent @RT(0) @T @F @DT @RT(4)DINT @RT(0) @T @T @BASIC 0 @F
@F @F
@T
@BEG_Attrib
0 @RT(1)1 @RT(32)lower limit for MoveId / MoveDir
@END_Attrib
1 1 @F @F @F @F

@Var @RT(9)cCompMold @RT(0) @T @F @DT @RT(4)DINT @RT(0) @T @T @BASIC 0 @F
@F @F
@T
@BEG_Attrib
0 @RT(3)101 @RT(14)Component Mold
@END_Attrib
1 1 @F @F @F @F

@Var @RT(12)cCompEjector @RT(0) @T @F @DT @RT(4)DINT @RT(0) @T @T @BASIC 0 @F
@F @F
@T
@BEG_Attrib
0 @RT(3)102 @RT(17)Component Ejector
@END_Attrib
1 1 @F @F @F @F

@Var @RT(18)cMoveBeginSequence @RT(0) @T @F @DT @RT(4)DINT @RT(0) @T @T @BASIC 0 @F
@F @F
@T
@BEG_Attrib
0 @RT(2)43 @RT(38)dummy movement for begin of a sequence
@END_Attrib
1 1 @F @F @F @F

@Var @RT(16)cMoveEndSequence @RT(0) @T @F @DT @RT(4)DINT @RT(0) @T @T @BASIC 0 @F
@F @F
@T
@BEG_Attrib
0 @RT(2)44 @RT(36)dummy movement for end of a sequence
@END_Attrib
1 1 @F @F @F @F

@Var @RT(14)cCompInjection @RT(0) @T @F @DT @RT(4)DINT @RT(0) @T @T @BASIC 0 @F
@F @F
@T
@BEG_Attrib
0 @RT(3)104 @RT(19)Component Injection
@END_Attrib
1 1 @F @F @F @F

@Var @RT(8)cMoveFwd @RT(0) @T @F @DT @RT(4)DINT @RT(0) @T @T @BASIC 0 @F
@F @F
@T
@BEG_Attrib
0 @RT(2)12 @RT(16)movement forward
@END_Attrib
1 1 @F @F @F @F

@Var @RT(8)cMoveBwd @RT(0) @T @F @DT @RT(4)DINT @RT(0) @T @T @BASIC 0 @F
@F @F
@T
@BEG_Attrib
0 @RT(2)11 @RT(17)movement backward
@END_Attrib
1 1 @F @F @F @F

@Var @RT(18)cMoveStartParallel @RT(0) @T @F @DT @RT(4)DINT @RT(0) @T @T @BASIC 0 @F
@F @F
@T
@BEG_Attrib
0 @RT(2)45 @RT(34)dummy movement for "StartParallel"
@END_Attrib
1 1 @F @F @F @F

@Var @RT(16)cMoveEndParallel @RT(0) @T @F @DT @RT(4)DINT @RT(0) @T @T @BASIC 0 @F
@F @F
@T
@BEG_Attrib
0 @RT(2)46 @RT(32)dummy movement for "EndParallel"
@END_Attrib
1 1 @F @F @F @F

@Var @RT(12)cMoveCooling @RT(0) @T @F @DT @RT(4)DINT @RT(0) @T @T @BASIC 0 @F
@F @F
@T
@BEG_Attrib
0 @RT(2)25 @RT(12)cooling time
@END_Attrib
1 1 @F @F @F @F

@Var @RT(10)cMoveShake @RT(0) @T @F @DT @RT(4)DINT @RT(0) @T @T @BASIC 0 @F
@F @F
@T
@BEG_Attrib
0 @RT(2)18 @RT(51)shaking movement (for example ejector vibrate mode)
@END_Attrib
1 1 @F @F @F @F

@Var @RT(8)cMoveOut @RT(0) @T @F @DT @RT(4)DINT @RT(0) @T @T @BASIC 0 @F
@F @F
@T
@BEG_Attrib
0 @RT(2)22 @RT(27)move out (for example core)
@END_Attrib
1 1 @F @F @F @F

@Var @RT(9)cMoveNone @RT(0) @T @F @DT @RT(4)DINT @RT(0) @T @T @BASIC 0 @F
@F @F
@T
@BEG_Attrib
0 @RT(13)cMinMoveIdent @RT(4)None
@END_Attrib
1 1 @F @F @F @F

@Var @RT(22)cODCDependencyDontCare @RT(0) @T @F @DT @RT(4)DINT @RT(0) @T @T @BASIC 0 @F
@F @F
@T
@BEG_Attrib
0 @RT(2)-1 @RT(76)dependency dont care, function unit not safety relevant, interpretation TRUE
@END_Attrib
1 1 @F @F @F @F

@Var @RT(9)cCompCore @RT(0) @T @F @DT @RT(4)DINT @RT(0) @T @T @BASIC 0 @F
@F @F
@T
@BEG_Attrib
0 @RT(3)109 @RT(14)Component Core
@END_Attrib
1 1 @F @F @F @F

@Var @RT(16)cMoveFwdInterPos @RT(0) @T @F @DT @RT(4)DINT @RT(0) @T @T @BASIC 0 @F
@F @F
@T
@BEG_Attrib
0 @RT(2)17 @RT(37)move forward to intermediate position
@END_Attrib
1 1 @F @F @F @F

@Var @RT(19)cMaxDeviceMovements @RT(0) @T @F @DT @RT(4)DINT @RT(0) @T @T @BASIC 0 @F
@F @F
@T
@BEG_Attrib
0 @RT(2)20 @RT(34)max number of movements per device
@END_Attrib
1 1 @F @F @F @F

@Var @RT(12)cMaxODCSteps @RT(0) @T @F @DT @RT(4)DINT @RT(0) @T @T @BASIC 0 @F
@F @F
@T
@BEG_Attrib
0 @RT(3)100 @RT(35)maximum number of rows in odc array
@END_Attrib
1 1 @F @F @F @F

@Var @RT(9)cCompNone @RT(0) @T @F @DT @RT(4)DINT @RT(0) @T @T @BASIC 0 @F
@F @F
@T
@BEG_Attrib
0 @RT(10)cMinCompId @RT(4)None
@END_Attrib
1 1 @F @F @F @F

@Var @RT(10)cMovePlast @RT(0) @T @F @DT @RT(4)DINT @RT(0) @T @T @BASIC 0 @F
@F @F
@T
@BEG_Attrib
0 @RT(2)13 @RT(23)plast movement (rotate)
@END_Attrib
1 1 @F @F @F @F

@Var @RT(17)cTimeOutSempahore @RT(0) @T @F @DT @RT(4)TIME @RT(0) @T @T @BASIC 0 @F
@F @F
@T
@BEG_Attrib
0 @RT(5)t#30s @RT(0)
@END_Attrib
1 1 @F @F @F @F

@Var @RT(19)cMaxStartConditions @RT(0) @T @F @DT @RT(4)DINT @RT(0) @T @T @BASIC 0 @F
@F @F
@T
@BEG_Attrib
0 @RT(2)10 @RT(51)max number of start condition steps in the sequence
@END_Attrib
1 1 @F @F @F @F

@Var @RT(18)cCompOperationMode @RT(0) @T @F @DT @RT(4)DINT @RT(0) @T @T @BASIC 0 @F
@F @F
@T
@BEG_Attrib
0 @RT(3)111 @RT(24)Component Operation Mode
@END_Attrib
1 1 @F @F @F @F

@Var @RT(24)cMoveIncreaseShotCounter @RT(0) @T @F @DT @RT(4)DINT @RT(0) @T @T @BASIC 0 @F
@F @F
@T
@BEG_Attrib
0 @RT(2)47 @RT(21)increase shot counter
@END_Attrib
1 1 @F @F @F @F

@Var @RT(25)cMaxMoveDevicesRegistered @RT(0) @T @F @DT @RT(4)DINT @RT(0) @T @T @BASIC 0 @F
@F @F
@T
@BEG_Attrib
0 @RT(2)50 @RT(49)max number of devices which are serving movements
@END_Attrib
1 1 @F @F @F @F

@Var @RT(19)cCycleTimeArraySize @RT(0) @T @F @DT @RT(4)DINT @RT(0) @T @T @BASIC 0 @F
@F @F
@T
@BEG_Attrib
0 @RT(1)3 @RT(48)size of array that contains the last cycle times
@END_Attrib
1 1 @F @F @F @F

@Var @RT(12)cAllDevIndex @RT(0) @T @F @DT @RT(4)DINT @RT(0) @T @T @BASIC 0 @F
@F @F
@T
@BEG_Attrib
0 @RT(2)11 @RT(59)to lock all devices of a component ( = cMaxDeviceIndex + 1)
@END_Attrib
1 1 @F @F @F @F

@Var @RT(19)cMoveStartCondition @RT(0) @T @F @DT @RT(4)DINT @RT(0) @T @T @BASIC 0 @F
@F @F
@T
@BEG_Attrib
0 @RT(2)52 @RT(35)dummy movement for "StartCondition"
@END_Attrib
1 1 @F @F @F @F

@Var @RT(10)cMinCompId @RT(0) @T @F @DT @RT(4)DINT @RT(0) @T @T @BASIC 0 @F
@F @F
@T
@BEG_Attrib
0 @RT(3)100 @RT(21)minimum Component ID
@END_Attrib
1 1 @F @F @F @F

@END_Const

@BEG_Export

@BEG_Kind
@ALGORITHM_BLOCK @RT(5)ABODC @STRUCTURED_TEXT
@RT(0) @RT(0) @RT(0)
@END_Kind

@BEG_Dcl
@RT(16)DclTreeContainer
110
@Var @RT(13)abInterpreter @RT(0) @T @T @DERIVED 0 @T @T @DT @RT(13)ABInterpreter @RT(0) @T @T @UNKNOWN 0 @F
@F @F
@T
@BEG_Attrib
3 @RT(0) @RT(0) @RT(0)
@END_Attrib
1 0 @F @F @F @F

@Var @RT(14)abKODC_Builder @RT(0) @T @T @DERIVED 0 @T @T @DT @RT(12)KODC_Builder @RT(0) @T @T @UNKNOWN 0 @F
@F @F
@T
@BEG_Attrib
3 @RT(0) @RT(0) @RT(0)
@END_Attrib
1 0 @F @F @F @F

@Var @RT(15)fbGetMoveNumber @RT(0) @T @T @DERIVED 0 @T @T @DT @RT(15)FBGetMoveNumber @RT(0) @T @T @UNKNOWN 0 @F
@F @F
@T
@BEG_Attrib
3 @RT(0) @RT(0) @RT(0)
@END_Attrib
1 0 @F @F @F @F

@Var @RT(12)fbAutoManual @RT(0) @T @T @DERIVED 0 @T @T @DT @RT(12)FBAutoManual @RT(0) @T @T @UNKNOWN 0 @F
@F @F
@T
@BEG_Attrib
3 @RT(0) @RT(0) @RT(0)
@END_Attrib
1 0 @F @F @F @F

@Var @RT(12)fbDebugTrace @RT(0) @T @T @DERIVED 0 @T @T @DT @RT(12)FBDebugTrace @RT(0) @T @T @UNKNOWN 0 @F
@F @F
@T
@BEG_Attrib
3 @RT(0) @RT(0) @RT(0)
@END_Attrib
1 0 @F @F @F @F

@Var @RT(12)g_SafetyData @RT(0) @T @T @DERIVED 0 @T @T @DT @RT(15)tsGlbSafetyData @RT(0) @T @T @UNKNOWN 0 @F
@F @F
@T
@BEG_Attrib
3 @RT(0) @RT(0) @RT(0)
@END_Attrib
1 6 @F @F @F @F

@Var @RT(13)fbDebugTrace2 @RT(0) @T @T @DERIVED 0 @T @T @DT @RT(13)FBDebugTrace2 @RT(0) @T @T @UNKNOWN 0 @F
@F @F
@T
@BEG_Attrib
3 @RT(0) @RT(0) @RT(0)
@END_Attrib
1 0 @F @F @F @F

@Var @RT(13)MovementsSema @RT(0) @T @T @DERIVED 0 @T @T @DT @RT(15)KRTOS_Semaphore @RT(0) @T @T @UNKNOWN 0 @F
@F @F
@T
@BEG_Attrib
3 @RT(0) @RT(34)protects sv_StartedManualMovements @RT(0)
@END_Attrib
1 5 @F @F @F @F

@Var @RT(14)sv_ODCSequence @RT(0) @T @T @DERIVED 0 @T @T @DT @RT(13)KODC_Sequence @RT(0) @T @T @UNKNOWN 0 @F
@F @F
@T
@BEG_Attrib
3 @RT(0) @RT(0) @RT(0)
@END_Attrib
1 8 @F @F @F @F

@Var @RT(17)sv_ODCSequenceInt @RT(0) @T @T @DERIVED 0 @T @T @DT @RT(21)tyODCSequenceInternal @RT(0) @T @T @UNKNOWN 0 @F
@F @F
@T
@BEG_Attrib
3 @RT(0) @RT(0) @RT(0)
@END_Attrib
1 8 @F @F @F @F

@Var @RT(15)sv_ODCMovements @RT(0) @T @T @DERIVED 0 @T @T @DT @RT(14)KODC_Movements @RT(0) @T @T @UNKNOWN 0 @F
@F @F
@T
@BEG_Attrib
3 @RT(0) @RT(0) @RT(0)
@END_Attrib
1 8 @F @F @F @F

@Var @RT(17)sv_dCycleDelaySet @RT(0) @T @F @DT @RT(4)TIME @RT(0) @T @T @BASIC 0 @F
@F @F
@T
@BEG_Attrib
3 @RT(0) @RT(0) @RT(0)
@END_Attrib
1 8 @F @F @F @F

@Var @RT(17)sv_dCycleDelayAct @RT(0) @T @F @DT @RT(4)TIME @RT(0) @T @T @BASIC 0 @F
@F @F
@T
@BEG_Attrib
3 @RT(0) @RT(0) @RT(0)
@END_Attrib
1 8 @F @F @F @F

@Var @RT(14)sv_bFirstCycle @RT(0) @T @F @DT @RT(4)BOOL @RT(0) @T @T @BASIC 0 @F
@F @F
@T
@BEG_Attrib
3 @RT(0) @RT(0) @RT(0)
@END_Attrib
1 8 @F @F @F @F

@Var @RT(12)sv_bInitDone @RT(0) @T @T @RENAMED 0 @T @T @DT @RT(4)BOOL @RT(0) @T @T @BASIC 0 @F
@F @F
@T
@BEG_Attrib
3 @RT(0) @RT(0) @RT(0)
@END_Attrib
1 8 @F @F @F @F

@Var @RT(29)sv_bCombinedMovementsInManual @RT(0) @T @T @RENAMED 0 @T @T @DT @RT(4)BOOL @RT(0) @T @T @BASIC 0 @F
@F @F
@T
@BEG_Attrib
3 @RT(0) @RT(0) @RT(0)
@END_Attrib
1 8 @F @F @F @F

@Var @RT(16)sv_OperationMode @RT(0) @T @T @RENAMED 0 @T @T @DT @RT(15)tnOperationMode @RT(0) @T @T @UNKNOWN 0 @F
@F @F
@T
@BEG_Attrib
3 @RT(0) @RT(0) @RT(0)
@END_Attrib
1 8 @F @F @F @F

@Var @RT(25)sv_StartedManualMovements @RT(0) @T @T @DERIVED 0 @T @T @DT @RT(28)tsStartedMoveDataODCExtended @RT(0) @T @T @UNKNOWN 0 @F
@F @F
@T
@BEG_Attrib
3 @RT(0) @RT(0) @RT(0)
@END_Attrib
1 8 @F @F @F @F

@Var @RT(21)sv_MovementsAvailable @RT(0) @T @T @DERIVED 0 @T @T @DT @RT(22)tyMovementRegisterList @RT(0) @T @T @UNKNOWN 0 @F
@F @F
@T
@BEG_Attrib
3 @RT(0) @RT(0) @RT(0)
@END_Attrib
1 8 @F @F @F @F

@Var @RT(19)sv_bODCFilesChanged @RT(0) @T @T @RENAMED 0 @T @T @DT @RT(4)BOOL @RT(0) @T @T @BASIC 0 @F
@F @F
@T
@BEG_Attrib
3 @RT(0) @RT(0) @RT(0)
@END_Attrib
1 8 @F @F @F @F

@Var @RT(24)sv_bProgramSwitchChanged @RT(0) @T @T @RENAMED 0 @T @T @DT @RT(4)BOOL @RT(0) @T @T @BASIC 0 @F
@F @F
@T
@BEG_Attrib
3 @RT(0) @RT(0) @RT(0)
@END_Attrib
1 8 @F @F @F @F

@Var @RT(21)sv_bActivationChanged @RT(0) @T @T @RENAMED 0 @T @T @DT @RT(4)BOOL @RT(0) @T @T @BASIC 0 @F
@F @F
@T
@BEG_Attrib
3 @RT(0) @RT(0) @RT(0)
@END_Attrib
1 8 @F @F @F @F

@Var @RT(19)sv_StartedMovements @RT(0) @T @T @DERIVED 0 @T @T @DT @RT(17)tsStartedMoveData @RT(0) @T @T @UNKNOWN 0 @F
@F @F
@T
@BEG_Attrib
3 @RT(0) @RT(0) @RT(0)
@END_Attrib
1 8 @F @F @F @F

@Var @RT(21)sv_ODCDeviceMovements @RT(0) @T @T @DERIVED 0 @T @T @DT @RT(23)tsODCDeviceMovementList @RT(0) @T @T @UNKNOWN 0 @F
@F @F
@T
@BEG_Attrib
3 @RT(0) @RT(57)list of all devices that registered movements for the ODC @RT(0)
@END_Attrib
1 8 @F @F @F @F

@Var @RT(22)sv_iMovementsAvailable @RT(0) @T @F @DT @RT(4)DINT @RT(0) @T @T @BASIC 0 @F
@F @F
@T
@BEG_Attrib
3 @RT(0) @RT(0) @RT(0)
@END_Attrib
1 8 @F @F @F @F

@Var @RT(20)sv_bAutoCycleRunning @RT(0) @T @F @DT @RT(4)BOOL @RT(0) @T @T @BASIC 0 @F
@F @F
@T
@BEG_Attrib
3 @RT(0) @RT(0) @RT(0)
@END_Attrib
1 8 @F @F @F @F

@Var @RT(16)sv_dMaxCycleTime @RT(0) @T @F @DT @RT(4)TIME @RT(0) @T @T @BASIC 0 @F
@F @F
@T
@BEG_Attrib
3 @RT(0) @RT(0) @RT(0)
@END_Attrib
1 8 @F @F @F @F

@Var @RT(13)sv_dCycleTime @RT(0) @T @F @DT @RT(4)TIME @RT(0) @T @T @BASIC 0 @F
@F @F
@T
@BEG_Attrib
3 @RT(0) @RT(0) @RT(0)
@END_Attrib
1 8 @F @F @F @F

@Var @RT(20)sv_dCycleTimeMachine @RT(0) @T @F @DT @RT(4)TIME @RT(0) @T @T @BASIC 0 @F
@F @F
@T
@BEG_Attrib
3 @RT(0) @RT(23)act. cylce time machine @RT(0)
@END_Attrib
1 8 @F @F @F @F

@Var @RT(26)sv_ODCSequenceGenerateTime @RT(0) @T @T @RENAMED 0 @T @T @DT @RT(13)DATE_AND_TIME @RT(0) @T @T @BASIC 0 @F
@F @F
@T
@BEG_Attrib
3 @RT(0) @RT(0) @RT(0)
@END_Attrib
1 8 @F @F @F @F

@Var @RT(20)sv_ODCSequenceBackup @RT(0) @T @T @DERIVED 0 @T @T @DT @RT(19)tyODCSequenceBackup @RT(0) @T @T @UNKNOWN 0 @F
@F @F
@T
@BEG_Attrib
3 @RT(0) @RT(0) @RT(0)
@END_Attrib
1 8 @F @F @F @F

@Var @RT(18)sv_iODCSequenceAct @RT(0) @T @T @RENAMED 0 @T @T @DT @RT(4)DINT @RT(0) @T @T @BASIC 0 @F
@F @F
@T
@BEG_Attrib
3 @RT(0) @RT(0) @RT(0)
@END_Attrib
1 8 @F @F @F @F

@Var @RT(21)sv_iSequenceToRestore @RT(0) @T @T @RENAMED 0 @T @T @DT @RT(4)DINT @RT(0) @T @T @BASIC 0 @F
@F @F
@T
@BEG_Attrib
3 @RT(0) @RT(0) @RT(0)
@END_Attrib
1 8 @F @F @F @F

@Var @RT(21)sv_ODCDescriptionPath @RT(0) @T @T @RENAMED 0 @T @T @DT @RT(11)STRING(255) @RT(0) @T @T @STRING 0 @F @RT(3)255 @F
@F @F
@T
@BEG_Attrib
3 @RT(0) @RT(0) @RT(0)
@END_Attrib
1 8 @F @F @F @F

@Var @RT(12)sv_DataState @RT(0) @T @T @RENAMED 0 @T @T @DT @RT(11)tnDataState @RT(0) @T @T @UNKNOWN 0 @F
@F @F
@T
@BEG_Attrib
3 @RT(0) @RT(0) @RT(0)
@END_Attrib
1 8 @F @F @F @F

@Var @RT(22)sv_iODCSequenceUpdated @RT(0) @T @F @DT @RT(4)DINT @RT(0) @T @T @BASIC 0 @F
@F @F
@T
@BEG_Attrib
3 @RT(0) @RT(0) @RT(0)
@END_Attrib
1 8 @F @F @F @F

@Var @RT(12)sv_iUsedRows @RT(0) @T @T @RENAMED 0 @T @T @DT @RT(4)DINT @RT(0) @T @T @BASIC 0 @F
@F @F
@T
@BEG_Attrib
3 @RT(0) @RT(0) @RT(0)
@END_Attrib
1 8 @F @F @F @F

@Var @RT(15)sv_iUsedColumns @RT(0) @T @T @RENAMED 0 @T @T @DT @RT(4)DINT @RT(0) @T @T @BASIC 0 @F
@F @F
@T
@BEG_Attrib
3 @RT(0) @RT(0) @RT(0)
@END_Attrib
1 8 @F @F @F @F

@Var @RT(10)sv_iInitOK @RT(0) @T @T @RENAMED 0 @T @T @DT @RT(4)DINT @RT(0) @T @T @BASIC 0 @F
@F @F
@T
@BEG_Attrib
3 @RT(0) @RT(92)0 nothing initialized, 10 sequence array initialized, 20 sequence array + safety initialized @RT(0)
@END_Attrib
1 8 @F @F @F @F

@Var @RT(13)evStopRequest @RT(0) @T @T @RENAMED 0 @T @T @DT @RT(14)tevStopRequest @RT(0) @T @T @UNKNOWN 0 @F
@F @F
@T
@BEG_Attrib
3 @RT(0) @RT(0) @RT(0)
@END_Attrib
1 7 @F @F @F @F

@Var @RT(16)evStartedStopped @RT(0) @T @T @RENAMED 0 @T @T @DT @RT(17)tevStartedStopped @RT(0) @T @T @UNKNOWN 0 @F
@F @F
@T
@BEG_Attrib
3 @RT(0) @RT(0) @RT(0)
@END_Attrib
1 7 @F @F @F @F

@Var @RT(14)evStartRequest @RT(0) @T @T @DERIVED 0 @T @T @DT @RT(15)tevStartRequest @RT(0) @T @T @UNKNOWN 0 @F
@F @F
@T
@BEG_Attrib
3 @RT(0) @RT(0) @RT(0)
@END_Attrib
1 7 @F @F @F @F

@Var @RT(25)evAlarmFinishCycleAndStop @RT(0) @T @T @DERIVED 0 @T @T @DT @RT(11)ALARM_EVENT @RT(0) @T @T @UNKNOWN 0 @F
@F @F
@T
@BEG_Attrib
3 @RT(0) @RT(0) @RT(0)
@END_Attrib
1 7 @F @F @F @F

@Var @RT(15)erODCInitFailed @RT(0) @T @T @RENAMED 0 @T @T @DT @RT(5)ALARM @RT(0) @T @T @BASIC 0 @F
@F @F
@T
@BEG_Attrib
3 @RT(0) @RT(0) @RT(0)
@END_Attrib
1 7 @F @F @F @F

@Var @RT(19)erCycleTimeExceeded @RT(0) @T @F @DT @RT(5)ALARM @RT(0) @T @T @BASIC 0 @F
@F @F
@T
@BEG_Attrib
3 @RT(0) @RT(0) @RT(0)
@END_Attrib
1 7 @F @F @F @F

@Var @RT(9)EV_Task_3 @RT(0) @T @F @DT @RT(4)TASK @RT(0) @T @T @BASIC 0 @F
@F @F
@T
@BEG_Attrib
3 @RT(0) @RT(0) @RT(0)
@END_Attrib
1 7 @F @F @F @F

@Var @RT(9)EV_Task_7 @RT(0) @T @T @RENAMED 0 @T @T @DT @RT(4)TASK @RT(0) @T @T @BASIC 0 @F
@F @F
@T
@BEG_Attrib
3 @RT(0) @RT(0) @RT(0)
@END_Attrib
1 7 @F @F @F @F

@Var @RT(9)PU_Task_3 @RT(0) @T @T @RENAMED 0 @T @T @DT @RT(4)TASK @RT(0) @T @T @BASIC 0 @F
@F @F
@T
@BEG_Attrib
3 @RT(0) @RT(0) @RT(0)
@END_Attrib
1 7 @F @F @F @F

@Var @RT(9)PU_Task_7 @RT(0) @T @T @RENAMED 0 @T @T @DT @RT(4)TASK @RT(0) @T @T @BASIC 0 @F
@F @F
@T
@BEG_Attrib
3 @RT(0) @RT(0) @RT(0)
@END_Attrib
1 7 @F @F @F @F

@Var @RT(10)TaskAnalog @RT(0) @T @F @DT @RT(4)TASK @RT(0) @T @T @BASIC 0 @F
@F @F
@T
@BEG_Attrib
3 @RT(0) @RT(0) @RT(0)
@END_Attrib
1 7 @F @F @F @F

@Var @RT(7)TaskMid @RT(0) @T @F @DT @RT(4)TASK @RT(0) @T @T @BASIC 0 @F
@F @F
@T
@BEG_Attrib
3 @RT(0) @RT(0) @RT(0)
@END_Attrib
1 7 @F @F @F @F

@Var @RT(8)erAssert @RT(0) @T @T @RENAMED 0 @T @T @DT @RT(5)ALARM @RT(0) @T @T @BASIC 0 @F
@F @F
@T
@BEG_Attrib
3 @RT(0) @RT(0) @RT(0)
@END_Attrib
1 7 @F @F @F @F

@Var @RT(5)dummy @RT(0) @T @F @DT @RT(4)DINT @RT(0) @T @T @BASIC 0 @F
@F @F
@T
@BEG_Attrib
3 @RT(0) @RT(0) @RT(0)
@END_Attrib
1 0 @F @F @F @F

@Var @RT(6)dummy2 @RT(0) @T @F @DT @RT(4)BOOL @RT(0) @T @T @BASIC 0 @F
@F @F
@T
@BEG_Attrib
3 @RT(0) @RT(0) @RT(0)
@END_Attrib
1 0 @F @F @F @F

@Var @RT(24)mStartedCombinedMovement @RT(0) @T @T @DERIVED 0 @T @T @DT @RT(17)tsStartedMoveInfo @RT(0) @T @T @UNKNOWN 0 @F
@F @F
@T
@BEG_Attrib
3 @RT(0) @RT(0) @RT(0)
@END_Attrib
1 0 @F @F @F @F

@Var @RT(11)mRecalcMode @RT(0) @T @T @DERIVED 0 @T @T @DT @RT(15)tnODCRecalcMode @RT(0) @T @T @UNKNOWN 0 @F
@F @F
@T
@BEG_Attrib
3 @RT(0) @RT(113)currently active recalc mode, set by aDoPendingRecalc when the ODC decided to start recalculation of the sequence @RT(0)
@END_Attrib
1 0 @F @F @F @F

@Var @RT(6)Status @RT(0) @T @T @DERIVED 0 @T @T @DT @RT(12)KRTOS_Status @RT(0) @T @T @UNKNOWN 0 @F
@F @F
@T
@BEG_Attrib
3 @RT(0) @RT(0) @RT(0)
@END_Attrib
1 0 @F @F @F @F

@Var @RT(11)mbStopCycle @RT(0) @T @F @DT @RT(4)BOOL @RT(0) @T @T @BASIC 0 @F
@F @F
@T
@BEG_Attrib
3 @RT(0) @RT(0) @RT(0)
@END_Attrib
1 0 @F @F @F @F

@Var @RT(16)mbStopAfterCycle @RT(0) @T @F @DT @RT(4)BOOL @RT(0) @T @T @BASIC 0 @F
@F @F
@T
@BEG_Attrib
3 @RT(0) @RT(0) @RT(0)
@END_Attrib
1 0 @F @F @F @F

@Var @RT(18)mbCycleTimeRunning @RT(0) @T @F @DT @RT(4)BOOL @RT(0) @T @T @BASIC 0 @F
@F @F
@T
@BEG_Attrib
3 @RT(0) @RT(0) @RT(0)
@END_Attrib
1 0 @F @F @F @F

@Var @RT(25)mbCycleTimeMachineRunning @RT(0) @T @F @DT @RT(4)BOOL @RT(0) @T @T @BASIC 0 @F
@F @F
@T
@BEG_Attrib
3 @RT(0) @RT(32)condition for cycle time machine @RT(0)
@END_Attrib
1 0 @F @F @F @F

@Var @RT(17)mbSequenceChanged @RT(0) @T @F @DT @RT(4)BOOL @RT(0) @T @T @BASIC 0 @F
@F @F
@T
@BEG_Attrib
3 @RT(0) @RT(74)the ODC sequence array possibly changed->need to backup when first started @RT(0)
@END_Attrib
1 0 @F @F @F @F

@Var @RT(27)mbIgnoreProgramSwitchChange @RT(0) @T @F @DT @RT(4)BOOL @RT(0) @T @T @BASIC 0 @F
@F @F
@T
@BEG_Attrib
3 @RT(0) @RT(68)ignore program switch or activation changes during mold data loading @RT(0)
@END_Attrib
1 0 @F @F @F @F

@Var @RT(14)mPendingRecalc @RT(0) @T @T @DERIVED 0 @T @T @DT @RT(15)tnODCRecalcMode @RT(0) @T @T @UNKNOWN 0 @F
@F @F
@T
@BEG_Attrib
3 @RT(0) @RT(65)recalculations requested by aSetPendingRecalc but not started yet @RT(0)
@END_Attrib
1 0 @F @F @F @F

@Var @RT(14)mbRecalcActive @RT(0) @T @F @DT @RT(4)BOOL @RT(0) @T @T @BASIC 0 @F
@F @F
@T
@BEG_Attrib
3 @RT(0) @RT(0) @RT(0)
@END_Attrib
1 0 @F @F @F @F

@Var @RT(8)TaskSlow @RT(0) @T @F @DT @RT(4)TASK @RT(0) @T @T @BASIC 0 @F
@F @F
@T
@BEG_Attrib
3 @RT(0) @RT(0) @RT(0)
@END_Attrib
1 7 @F @F @F @F

@Var @RT(17)sv_iActiveEditors @RT(0) @T @T @RENAMED 0 @T @T @DT @RT(4)DINT @RT(0) @T @T @BASIC 0 @F
@F @F
@T
@BEG_Attrib
3 @RT(0) @RT(0) @RT(0)
@END_Attrib
1 8 @F @F @F @F

@Var @RT(29)sv_StartConditionInstanceData @RT(0) @T @T @DERIVED 0 @T @T @DT @RT(23)tyStartCondInstanceData @RT(0) @T @T @UNKNOWN 0 @F
@F @F
@T
@BEG_Attrib
3 @RT(0) @RT(50)list with start condition params for all instances @RT(0)
@END_Attrib
1 8 @F @F @F @F

@Var @RT(26)erCompNotInCorrectPosition @RT(0) @T @F @DT @RT(5)ALARM @RT(0) @T @T @BASIC 0 @F
@F @F
@T
@BEG_Attrib
3 @RT(0) @RT(0) @RT(0)
@END_Attrib
1 7 @F @F @F @F

@Var @RT(22)sv_bUseProgramSwitches @RT(0) @T @F @DT @RT(4)BOOL @RT(0) @T @T @BASIC 0 @F
@F @F
@T
@BEG_Attrib
3 @RT(0) @RT(84)TRUE: create sequence by using program switches; FALSE: use sequence from ODC editor @RT(0)
@END_Attrib
1 8 @F @F @F @F

@Var @RT(17)erTeachModeActive @RT(0) @T @F @DT @RT(5)ALARM @RT(0) @T @T @BASIC 0 @F
@F @F
@T
@BEG_Attrib
3 @RT(0) @RT(0) @RT(0)
@END_Attrib
1 7 @F @F @F @F

@Var @RT(15)evCheckLocklist @RT(0) @T @T @RENAMED 0 @T @T @DT @RT(16)tevCheckLocklist @RT(0) @T @T @UNKNOWN 0 @F
@F @F
@T
@BEG_Attrib
3 @RT(0) @RT(0) @RT(0)
@END_Attrib
1 7 @F @F @F @F

@Var @RT(13)sv_TraceLevel @RT(0) @T @T @DERIVED 0 @T @T @DT @RT(12)tsTraceLevel @RT(0) @T @T @UNKNOWN 0 @F
@F @F
@T
@BEG_Attrib
3 @RT(0) @RT(0) @RT(0)
@END_Attrib
1 8 @F @F @F @F

@Var @RT(23)sv_dCalculatedCycleTime @RT(0) @T @F @DT @RT(4)TIME @RT(0) @T @T @BASIC 0 @F
@F @F
@T
@BEG_Attrib
3 @RT(0) @RT(52)calculated cycle time (written by machine sequencer) @RT(0)
@END_Attrib
1 8 @F @F @F @F

@Var @RT(27)sv_iEditorPropertiesChanged @RT(0) @T @F @DT @RT(4)DINT @RT(0) @T @T @BASIC 0 @F
@F @F
@T
@BEG_Attrib
3 @RT(0) @RT(0) @RT(0)
@END_Attrib
1 8 @F @F @F @F

@Var @RT(25)sv_dAllowedCycleDeviation @RT(0) @T @F @DT @RT(4)TIME @RT(0) @T @T @BASIC 0 @F
@F @F
@T
@BEG_Attrib
3 @RT(0) @RT(0) @RT(0)
@END_Attrib
1 8 @F @F @F @F

@Var @RT(13)TaskSequencer @RT(0) @T @T @RENAMED 0 @T @T @DT @RT(4)TASK @RT(0) @T @T @BASIC 0 @F
@F @F
@T
@BEG_Attrib
3 @RT(0) @RT(0) @RT(0)
@END_Attrib
1 7 @F @F @F @F

@Var @RT(30)erMovementDuringActiveSequence @RT(0) @T @F @DT @RT(5)ALARM @RT(0) @T @T @BASIC 0 @F
@F @F
@T
@BEG_Attrib
3 @RT(0) @RT(0) @RT(0)
@END_Attrib
1 7 @F @F @F @F

@Var @RT(30)erSequenceDuringActiveMovement @RT(0) @T @F @DT @RT(5)ALARM @RT(0) @T @T @BASIC 0 @F
@F @F
@T
@BEG_Attrib
3 @RT(0) @RT(0) @RT(0)
@END_Attrib
1 7 @F @F @F @F

@Var @RT(27)erMachineSequenceNotCreated @RT(0) @T @F @DT @RT(5)ALARM @RT(0) @T @T @BASIC 0 @F
@F @F
@T
@BEG_Attrib
3 @RT(0) @RT(0) @RT(0)
@END_Attrib
1 7 @F @F @F @F

@Var @RT(17)sv_dLastCycleTime @RT(0) @T @F @DT @RT(4)TIME @RT(0) @T @T @BASIC 0 @F
@F @F
@T
@BEG_Attrib
3 @RT(0) @RT(0) @RT(0)
@END_Attrib
1 8 @F @F @F @F

@Var @RT(8)sv_bTRUE @RT(0) @T @F @DT @RT(4)BOOL @RT(0) @T @T @BASIC 0 @F
@F @F
@T
@BEG_Attrib
3 @RT(0) @RT(0) @RT(0)
@END_Attrib
1 8 @F @F @F @F

@Var @RT(20)mbEjeBwdAtCycleStart @RT(0) @T @F @DT @RT(4)BOOL @RT(0) @T @T @BASIC 0 @F
@F @F
@T
@BEG_Attrib
3 @RT(0) @RT(97)info if ejector must be bwd at the beginning of the cycle (taken from safety array of first step) @RT(0)
@END_Attrib
1 0 @F @F @F @F

@Var @RT(27)miIndexEjectorInSafetyArray @RT(0) @T @F @DT @RT(4)DINT @RT(0) @T @T @BASIC 0 @F
@F @F
@T
@BEG_Attrib
3 @RT(0) @RT(0) @RT(0)
@END_Attrib
1 0 @F @F @F @F

@Var @RT(25)sv_bODCCombinedMoveActive @RT(0) @T @F @DT @RT(4)BOOL @RT(0) @T @T @BASIC 0 @F
@F @F
@T
@BEG_Attrib
3 @RT(0) @RT(87)TRUE: combined movement (for example closing sequence) is active (only in manual mode!) @RT(0)
@END_Attrib
1 8 @F @F @F @F

@Var @RT(23)mStartConditionPosArray @RT(0) @T @T @DERIVED 0 @T @T @DT @RT(24)tyStartConditionPosArray @RT(0) @T @T @UNKNOWN 0 @F
@F @F
@T
@BEG_Attrib
3 @RT(0) @RT(90)array with information about the position of each start condition in the internal sequence @RT(0)
@END_Attrib
1 0 @F @F @F @F

@Var @RT(11)sv_DeviceId @RT(0) @T @T @DERIVED 0 @T @T @DT @RT(10)tsDeviceId @RT(0) @T @T @UNKNOWN 0 @F
@F @F
@T
@BEG_Attrib
3 @RT(0) @RT(0) @RT(0)
@END_Attrib
1 8 @F @F @F @F

@Var @RT(22)sv_bOverrideCoreSafety @RT(0) @T @F @DT @RT(4)BOOL @RT(0) @T @T @BASIC 0 @F
@F @F
@T
@BEG_Attrib
3 @RT(0) @RT(0) @RT(0)
@END_Attrib
1 8 @F @F @F @F

@Var @RT(25)sv_bOverrideEjectorSafety @RT(0) @T @F @DT @RT(4)BOOL @RT(0) @T @T @BASIC 0 @F
@F @F
@T
@BEG_Attrib
3 @RT(0) @RT(0) @RT(0)
@END_Attrib
1 8 @F @F @F @F

@Var @RT(17)sv_ActiveSequence @RT(0) @T @T @DERIVED 0 @T @T @DT @RT(16)tsActiveSequence @RT(0) @T @T @UNKNOWN 0 @F
@F @F
@T
@BEG_Attrib
3 @RT(0) @RT(0) @RT(0)
@END_Attrib
1 8 @F @F @F @F

@Var @RT(16)sv_LoopParameter @RT(0) @T @T @DERIVED 0 @T @T @DT @RT(10)tyLoopData @RT(0) @T @T @UNKNOWN 0 @F
@F @F
@T
@BEG_Attrib
3 @RT(0) @RT(39)array with data of all programmed loops @RT(0)
@END_Attrib
1 8 @F @F @F @F

@Var @RT(25)g_iAutoCycleLoopStartLine @RT(0) @T @F @DT @RT(4)DINT @RT(0) @T @T @BASIC 0 @F
@F @F
@T
@BEG_Attrib
3 @RT(0) @RT(0) @RT(0)
@END_Attrib
1 6 @F @F @F @F

@Var @RT(23)g_iAutoCycleLoopEndLine @RT(0) @T @F @DT @RT(4)DINT @RT(0) @T @T @BASIC 0 @F
@F @F
@T
@BEG_Attrib
3 @RT(0) @RT(0) @RT(0)
@END_Attrib
1 6 @F @F @F @F

@Var @RT(26)sv_InterpreterParallelInfo @RT(0) @T @T @DERIVED 0 @T @T @DT @RT(17)tyODCParallelInfo @RT(0) @T @T @UNKNOWN 0 @F
@F @F
@T
@BEG_Attrib
3 @RT(0) @RT(61)internal state information of the interpreter, useful for HMI @RT(0)
@END_Attrib
1 8 @F @F @F @F

@Var @RT(27)g_iODCMoveDevicesRegistered @RT(0) @T @F @DT @RT(4)DINT @RT(0) @T @T @BASIC 0 @F
@F @F
@T
@BEG_Attrib
3 @RT(0) @RT(48)number of registered devices with ODC movements  @RT(0)
@END_Attrib
1 6 @F @F @F @F

@Var @RT(24)sv_bSequenceInterruption @RT(0) @T @F @DT @RT(4)BOOL @RT(0) @T @T @BASIC 0 @F
@F @F
@T
@BEG_Attrib
3 @RT(0) @RT(29)TRUE: sequence is interrupted @RT(0)
@END_Attrib
1 8 @F @F @F @F

@Var @RT(10)di_StepFwd @RT(0) @T @T @RENAMED 0 @T @T @DT @RT(4)BOOL @RT(0) @T @T @BASIC 0 @F
@F @F
@T
@BEG_Attrib
3 @RT(0) @RT(0) @RT(0)
@END_Attrib
1 8 @F @F @F @F

@Var @RT(10)di_StepBwd @RT(0) @T @T @RENAMED 0 @T @T @DT @RT(4)BOOL @RT(0) @T @T @BASIC 0 @F
@F @F
@T
@BEG_Attrib
3 @RT(0) @RT(0) @RT(0)
@END_Attrib
1 8 @F @F @F @F

@Var @RT(10)PU_Task_13 @RT(0) @T @T @RENAMED 0 @T @T @DT @RT(4)TASK @RT(0) @T @T @BASIC 0 @F
@F @F
@T
@BEG_Attrib
3 @RT(0) @RT(0) @RT(0)
@END_Attrib
1 7 @F @F @F @F

@Var @RT(23)mActiveStepBwdMovements @RT(0) @T @T @DERIVED 0 @T @T @DT @RT(18)tyStepBwdMovements @RT(0) @T @T @UNKNOWN 0 @F
@F @F
@T
@BEG_Attrib
3 @RT(0) @RT(27)ArrayIndex = column number! @RT(0)
@END_Attrib
1 0 @F @F @F @F

@Var @RT(19)erNoInverseMovement @RT(0) @T @F @DT @RT(5)ALARM @RT(0) @T @T @BASIC 0 @F
@F @F
@T
@BEG_Attrib
3 @RT(0) @RT(0) @RT(0)
@END_Attrib
1 7 @F @F @F @F

@Var @RT(17)sv_bStepBwdActive @RT(0) @T @F @DT @RT(4)BOOL @RT(0) @T @T @BASIC 0 @F
@F @F
@T
@BEG_Attrib
3 @RT(0) @RT(28)TRUE: stepping bwd is active @RT(0)
@END_Attrib
1 8 @F @F @F @F

@Var @RT(22)erTooManyStartParallel @RT(0) @T @F @DT @RT(5)ALARM @RT(0) @T @T @BASIC 0 @F
@F @F
@T
@BEG_Attrib
3 @RT(0) @RT(0) @RT(0)
@END_Attrib
1 7 @F @F @F @F

@Var @RT(20)sv_SequenceDimension @RT(0) @T @T @DERIVED 0 @T @T @DT @RT(19)tsSequenceDimension @RT(0) @T @T @UNKNOWN 0 @F
@F @F
@T
@BEG_Attrib
3 @RT(0) @RT(47)contains the maximum size of the sequence array @RT(0)
@END_Attrib
1 8 @F @F @F @F

@Var @RT(10)TaskInject @RT(0) @T @T @RENAMED 0 @T @T @DT @RT(4)TASK @RT(0) @T @T @BASIC 0 @F
@F @F
@T
@BEG_Attrib
3 @RT(0) @RT(0) @RT(0)
@END_Attrib
1 7 @F @F @F @F

@Var @RT(27)evModifyCycleStartCondition @RT(0) @T @T @DERIVED 0 @T @T @DT @RT(28)tevModifyCycleStartCondition @RT(0) @T @T @UNKNOWN 0 @F
@F @F
@T
@BEG_Attrib
3 @RT(0) @RT(0) @RT(0)
@END_Attrib
1 7 @F @F @F @F

@Var @RT(25)sv_bRecalcPendingOrActive @RT(0) @T @F @DT @RT(4)BOOL @RT(0) @T @T @BASIC 0 @F
@F @F
@T
@BEG_Attrib
3 @RT(0) @RT(169)The ODC wants to recalc the sequence or a recalc is currently active. Any evStartRequest sent at this time can potentially be ignored if recalculation is already active. @RT(0)
@END_Attrib
1 8 @F @F @F @F

@Var @RT(16)mbResetCycleTime @RT(0) @T @F @DT @RT(4)BOOL @RT(0) @T @T @BASIC 0 @F
@F @F
@T
@BEG_Attrib
3 @RT(0) @RT(0) @RT(0)
@END_Attrib
1 0 @F @F @F @F

@Var @RT(23)mbResetCycleTimeMachine @RT(0) @T @F @DT @RT(4)BOOL @RT(0) @T @T @BASIC 0 @F
@F @F
@T
@BEG_Attrib
3 @RT(0) @RT(0) @RT(0)
@END_Attrib
1 0 @F @F @F @F

@Var @RT(17)evNewCycleStarted @RT(0) @T @T @DERIVED 0 @T @T @DT @RT(13)tevCycleStart @RT(0) @T @T @UNKNOWN 0 @F
@F @F
@T
@BEG_Attrib
3 @RT(0) @RT(0) @RT(0)
@END_Attrib
1 7 @F @F @F @F

@END_Dcl

@END_Export

@BEG_Body

41

@BEG_Export

@BEG_Algo
@ALGORITHM @RT(18)aIsAnyColumnActive @STRUCTURED_TEXT
@RT(0) @RT(0) @RT(0) @F @F
@END_Algo

@BEG_Dcl
@RT(16)DclTreeContainer
2
@Var @RT(7)bActive @RT(0) @T @F @DT @RT(4)BOOL @RT(0) @T @T @BASIC 0 @F
@F @F
@T
@BEG_Attrib
3 @RT(0) @RT(0) @RT(0)
@END_Attrib
1 3 @F @F @F @F

@Var @RT(1)i @RT(0) @T @F @DT @RT(4)DINT @RT(0) @T @T @BASIC 0 @F
@F @F
@T
@BEG_Attrib
3 @RT(0) @RT(0) @RT(0)
@END_Attrib
1 4 @F @F @F @F

@END_Dcl

@END_Export

@BEG_Export

@BEG_Algo
@ALGORITHM @RT(15)aCheckCycleTime @STRUCTURED_TEXT
@RT(0) @RT(0) @RT(0) @F @F
@END_Algo

@BEG_Dcl
@RT(16)DclTreeContainer
4
@Var @RT(14)CycleTimeArray @RT(0) @T @T @DERIVED 0 @T @T @DT @RT(11)tyCycleTime @RT(0) @T @T @UNKNOWN 0 @F
@F @F
@T
@BEG_Attrib
3 @RT(0) @RT(0) @RT(0)
@END_Attrib
1 0 @F @F @F @F

@Var @RT(1)i @RT(0) @T @F @DT @RT(4)DINT @RT(0) @T @T @BASIC 0 @F
@F @F
@T
@BEG_Attrib
3 @RT(1)1 @RT(0) @RT(0)
@END_Attrib
1 0 @F @F @F @F

@Var @RT(4)dSum @RT(0) @T @F @DT @RT(4)TIME @RT(0) @T @T @BASIC 0 @F
@F @F
@T
@BEG_Attrib
3 @RT(0) @RT(0) @RT(0)
@END_Attrib
1 0 @F @F @F @F

@Var @RT(17)dAverageCycleTime @RT(0) @T @F @DT @RT(4)TIME @RT(0) @T @T @BASIC 0 @F
@F @F
@T
@BEG_Attrib
3 @RT(0) @RT(0) @RT(0)
@END_Attrib
1 0 @F @F @F @F

@END_Dcl

@END_Export

@BEG_Export

@BEG_Algo
@PROCESS_ALGORITHM @RT(16)paBackupSequence @STRUCTURED_TEXT
@RT(0) @RT(0) @RT(8)TaskSlow @F @F
@END_Algo

@BEG_Dcl
@RT(16)DclTreeContainer
0
@END_Dcl

@END_Export

@BEG_Export

@BEG_Algo
@ALGORITHM @RT(17)aSetPendingRecalc @STRUCTURED_TEXT
@RT(0) @RT(0) @RT(0) @F @F
@END_Algo

@BEG_Dcl
@RT(16)DclTreeContainer
1
@Var @RT(10)RecalcMode @RT(0) @T @T @DERIVED 0 @T @T @DT @RT(15)tnODCRecalcMode @RT(0) @T @T @UNKNOWN 0 @F
@F @F
@T
@BEG_Attrib
3 @RT(0) @RT(40)How much of the ODC array to recalculate @RT(0)
@END_Attrib
1 1 @F @F @F @F

@END_Dcl

@END_Export

@BEG_Export

@BEG_Algo
@ALGORITHM @RT(16)aDoPendingRecalc @STRUCTURED_TEXT
@RT(0) @RT(0) @RT(0) @F @F
@END_Algo

@BEG_Dcl
@RT(16)DclTreeContainer
1
@Var @RT(14)bStartedRecalc @RT(0) @T @F @DT @RT(4)BOOL @RT(0) @T @T @BASIC 0 @F
@F @F
@T
@BEG_Attrib
3 @RT(0) @RT(0) @RT(0)
@END_Attrib
1 3 @F @F @F @F

@END_Dcl

@END_Export

@BEG_Export

@BEG_Algo
@PROCESS_ALGORITHM @RT(14)paInitSequence @SEQUENTIAL_FLOW_CHART
@RT(0) @RT(0) @RT(7)TaskMid @F @F
@END_Algo

@BEG_Dcl
@RT(16)DclTreeContainer
34
@Var @RT(11)iCalledInit @RT(0) @T @F @DT @RT(4)DINT @RT(0) @T @T @BASIC 0 @F
@F @F
@T
@BEG_Attrib
3 @RT(0) @RT(0) @RT(0)
@END_Attrib
1 0 @F @F @F @F

@Var @RT(13)iCalledCreate @RT(0) @T @F @DT @RT(4)DINT @RT(0) @T @T @BASIC 0 @F
@F @F
@T
@BEG_Attrib
3 @RT(0) @RT(0) @RT(0)
@END_Attrib
1 0 @F @F @F @F

@Var @RT(7)iTmpRow @RT(0) @T @F @DT @RT(4)DINT @RT(0) @T @T @BASIC 0 @F
@F @F
@T
@BEG_Attrib
3 @RT(0) @RT(0) @RT(0)
@END_Attrib
1 4 @F @F @F @F

@Var @RT(7)iTmpCol @RT(0) @T @F @DT @RT(4)DINT @RT(0) @T @T @BASIC 0 @F
@F @F
@T
@BEG_Attrib
3 @RT(0) @RT(0) @RT(0)
@END_Attrib
1 4 @F @F @F @F

@Var @RT(5)iMove @RT(0) @T @F @DT @RT(4)DINT @RT(0) @T @T @BASIC 0 @F
@F @F
@T
@BEG_Attrib
3 @RT(0) @RT(0) @RT(0)
@END_Attrib
1 4 @F @F @F @F

@Var @RT(7)iDevice @RT(0) @T @F @DT @RT(4)DINT @RT(0) @T @T @BASIC 0 @F
@F @F
@T
@BEG_Attrib
3 @RT(0) @RT(0) @RT(0)
@END_Attrib
1 4 @F @F @F @F

@Var @RT(9)bInitDone @RT(0) @T @F @DT @RT(4)BOOL @RT(0) @T @T @BASIC 0 @F
@F @F
@T
@BEG_Attrib
3 @RT(0) @RT(0) @RT(0)
@END_Attrib
1 0 @F @F @F @F

@Var @RT(18)abSequDependencies @RT(0) @T @T @DERIVED 0 @T @T @DT @RT(18)ABSequDependencies @RT(0) @T @T @UNKNOWN 0 @F
@F @F
@T
@BEG_Attrib
3 @RT(0) @RT(0) @RT(0)
@END_Attrib
1 0 @F @F @F @F

@Var @RT(5)fbRTC @RT(0) @T @T @DERIVED 0 @T @T @DT @RT(3)RTC @RT(0) @T @T @UNKNOWN 0 @F
@F @F
@T
@BEG_Attrib
3 @RT(0) @RT(0) @RT(0)
@END_Attrib
1 0 @F @F @F @F

@Var @RT(6)bError @RT(0) @T @F @DT @RT(4)BOOL @RT(0) @T @T @BASIC 0 @F
@F @F
@T
@BEG_Attrib
3 @RT(0) @RT(0) @RT(0)
@END_Attrib
1 0 @F @F @F @F

@Var @RT(10)RecalcMode @RT(0) @T @T @DERIVED 0 @T @T @DT @RT(15)tnODCRecalcMode @RT(0) @T @T @UNKNOWN 0 @F
@F @F
@T
@BEG_Attrib
3 @RT(0) @RT(0) @RT(0)
@END_Attrib
1 0 @F @F @F @F

@Var @RT(18)EmptySequenceEntry @RT(0) @T @T @DERIVED 0 @T @T @DT @RT(9)KODC_Step @RT(0) @T @T @UNKNOWN 0 @F
@F @F
@T
@BEG_Attrib
3 @RT(81)(iCompId:=cCompNone,iMoveDir:=cMoveNone,iMoveId:=cMoveNone,iIndexId:=1,iCount:=0) @RT(0) @RT(0)
@END_Attrib
1 15 @F @F @F @F

@Var @RT(5)sPath @RT(0) @T @F @DT @RT(11)STRING(255) @RT(0) @T @T @STRING 0 @F @RT(3)255 @F
@F @F
@T
@BEG_Attrib
3 @RT(0) @RT(0) @RT(0)
@END_Attrib
1 0 @F @F @F @F

@Var @RT(10)bFirstCall @RT(0) @T @F @DT @RT(4)BOOL @RT(0) @T @T @BASIC 0 @F
@F @F
@T
@BEG_Attrib
3 @RT(0) @RT(0) @RT(0)
@END_Attrib
1 0 @F @F @F @F

@Var @RT(9)sWorkPath @RT(0) @T @F @DT @RT(11)STRING(255) @RT(0) @T @T @STRING 0 @F @RT(3)255 @F
@F @F
@T
@BEG_Attrib
3 @RT(0) @RT(0) @RT(0)
@END_Attrib
1 0 @F @F @F @F

@Var @RT(1)k @RT(0) @T @F @DT @RT(4)DINT @RT(0) @T @T @BASIC 0 @F
@F @F
@T
@BEG_Attrib
3 @RT(0) @RT(0) @RT(0)
@END_Attrib
1 4 @F @F @F @F

@Var @RT(9)iInstance @RT(0) @T @F @DT @RT(4)DINT @RT(0) @T @T @BASIC 0 @F
@F @F
@T
@BEG_Attrib
3 @RT(0) @RT(0) @RT(0)
@END_Attrib
1 0 @F @F @F @F

@Var @RT(15)fbLockUnlockAll @RT(0) @T @T @DERIVED 0 @T @T @DT @RT(12)FBLockUnlock @RT(0) @T @T @UNKNOWN 0 @F
@F @F
@T
@BEG_Attrib
3 @RT(87)(DeviceId:=(CompId:=cCompAll,IndexId:=cAllDevIndex),MoveDir:=cMoveAll,MoveId:=cMoveAll) @RT(0) @RT(0)
@END_Attrib
1 0 @F @F @F @F

@Var @RT(8)DeviceId @RT(0) @T @T @DERIVED 0 @T @T @DT @RT(10)tsDeviceId @RT(0) @T @T @UNKNOWN 0 @F
@F @F
@T
@BEG_Attrib
3 @RT(0) @RT(0) @RT(0)
@END_Attrib
1 0 @F @F @F @F

@Var @RT(1)i @RT(0) @T @F @DT @RT(4)DINT @RT(0) @T @T @BASIC 0 @F
@F @F
@T
@BEG_Attrib
3 @RT(0) @RT(0) @RT(0)
@END_Attrib
1 4 @F @F @F @F

@Var @RT(9)bTryAgain @RT(0) @T @F @DT @RT(4)BOOL @RT(0) @T @T @BASIC 0 @F
@F @F
@T
@BEG_Attrib
3 @RT(0) @RT(0) @RT(0)
@END_Attrib
1 0 @F @F @F @F

@Var @RT(12)FailedRecalc @RT(0) @T @T @DERIVED 0 @T @T @DT @RT(15)tnODCRecalcMode @RT(0) @T @T @UNKNOWN 0 @F
@F @F
@T
@BEG_Attrib
3 @RT(0) @RT(0) @RT(0)
@END_Attrib
1 0 @F @F @F @F

@Var @RT(6)iCount @RT(0) @T @F @DT @RT(3)INT @RT(0) @T @T @BASIC 0 @F
@F @F
@T
@BEG_Attrib
3 @RT(0) @RT(0) @RT(0)
@END_Attrib
1 0 @F @F @F @F

@Var @RT(12)iOrigEndLine @RT(0) @T @F @DT @RT(4)DINT @RT(0) @T @T @BASIC 0 @F
@F @F
@T
@BEG_Attrib
3 @RT(0) @RT(0) @RT(0)
@END_Attrib
1 0 @F @F @F @F

@Var @RT(13)StepBeginLoop @RT(0) @T @T @DERIVED 0 @T @T @DT @RT(9)KODC_Step @RT(0) @T @T @UNKNOWN 0 @F
@F @F
@T
@BEG_Attrib
3 @RT(85)(iCompId:=cCompODC,iMoveDir:=cMoveNone,iMoveId:=cMoveBeginLoop,iIndexId:=1,iCount:=1) @RT(0) @RT(0)
@END_Attrib
1 0 @F @F @F @F

@Var @RT(11)StepEndLoop @RT(0) @T @T @DERIVED 0 @T @T @DT @RT(9)KODC_Step @RT(0) @T @T @UNKNOWN 0 @F
@F @F
@T
@BEG_Attrib
3 @RT(83)(iCompId:=cCompODC,iMoveDir:=cMoveNone,iMoveId:=cMoveEndLoop,iIndexId:=1,iCount:=1) @RT(0) @RT(0)
@END_Attrib
1 0 @F @F @F @F

@Var @RT(8)iTmpCol2 @RT(0) @T @F @DT @RT(4)DINT @RT(0) @T @T @BASIC 0 @F
@F @F
@T
@BEG_Attrib
3 @RT(0) @RT(6)column @RT(0)
@END_Attrib
1 4 @F @F @F @F

@Var @RT(8)iTmpRow2 @RT(0) @T @F @DT @RT(4)DINT @RT(0) @T @T @BASIC 0 @F
@F @F
@T
@BEG_Attrib
3 @RT(0) @RT(4)line @RT(0)
@END_Attrib
1 4 @F @F @F @F

@Var @RT(8)bAddLoop @RT(0) @T @F @DT @RT(4)BOOL @RT(0) @T @T @BASIC 0 @F
@F @F
@T
@BEG_Attrib
3 @RT(0) @RT(0) @RT(0)
@END_Attrib
1 0 @F @F @F @F

@Var @RT(4)iTmp @RT(0) @T @F @DT @RT(4)DINT @RT(0) @T @T @BASIC 0 @F
@F @F
@T
@BEG_Attrib
3 @RT(0) @RT(0) @RT(0)
@END_Attrib
1 0 @F @F @F @F

@Var @RT(16)DeviceIdEjector1 @RT(0) @T @T @DERIVED 0 @T @T @DT @RT(10)tsDeviceId @RT(0) @T @T @UNKNOWN 0 @F
@F @F
@T
@BEG_Attrib
3 @RT(33)(CompId:=cCompEjector,IndexId:=1) @RT(0) @RT(0)
@END_Attrib
1 0 @F @F @F @F

@Var @RT(20)DependencyEjectorBwd @RT(0) @T @F @DT @RT(5)LWORD @RT(0) @T @T @BASIC 0 @F
@F @F
@T
@BEG_Attrib
3 @RT(0) @RT(41)dependency which represents "ejector bwd" @RT(0)
@END_Attrib
1 0 @F @F @F @F

@Var @RT(5)bInit @RT(0) @T @F @DT @RT(4)BOOL @RT(0) @T @T @BASIC 0 @F
@F @F
@T
@BEG_Attrib
3 @RT(0) @RT(0) @RT(0)
@END_Attrib
1 0 @F @F @F @F

@Var @RT(18)iNoOfStartParallel @RT(0) @T @F @DT @RT(4)DINT @RT(0) @T @T @BASIC 0 @F
@F @F
@T
@BEG_Attrib
3 @RT(0) @RT(0) @RT(0)
@END_Attrib
1 0 @F @F @F @F

@END_Dcl

@END_Export

@BEG_Export

@BEG_Algo
@ALGORITHM @RT(15)aClearStepState @STRUCTURED_TEXT
@RT(0) @RT(0) @RT(0) @F @F
@END_Algo

@BEG_Dcl
@RT(16)DclTreeContainer
4
@Var @RT(14)fbSetStepState @RT(0) @T @T @DERIVED 0 @T @T @DT @RT(14)FBSetStepState @RT(0) @T @T @UNKNOWN 0 @F
@F @F
@T
@BEG_Attrib
3 @RT(0) @RT(0) @RT(0)
@END_Attrib
1 0 @F @F @F @F

@Var @RT(7)iTmpRow @RT(0) @T @F @DT @RT(4)DINT @RT(0) @T @T @BASIC 0 @F
@F @F
@T
@BEG_Attrib
3 @RT(0) @RT(0) @RT(0)
@END_Attrib
1 4 @F @F @F @F

@Var @RT(10)iTmpColumn @RT(0) @T @F @DT @RT(4)DINT @RT(0) @T @T @BASIC 0 @F
@F @F
@T
@BEG_Attrib
3 @RT(0) @RT(0) @RT(0)
@END_Attrib
1 4 @F @F @F @F

@Var @RT(21)bExcludeActiveColumns @RT(0) @T @F @DT @RT(4)BOOL @RT(0) @T @T @BASIC 0 @F
@F @F
@T
@BEG_Attrib
3 @RT(0) @RT(0) @RT(0)
@END_Attrib
1 1 @F @F @F @F

@END_Dcl

@END_Export

@BEG_Export

@BEG_Algo
@ALGORITHM @RT(24)aStartAndCheckConditions @STRUCTURED_TEXT
@RT(0) @RT(0) @RT(0) @F @F
@END_Algo

@BEG_Dcl
@RT(16)DclTreeContainer
9
@Var @RT(7)StepPos @RT(0) @T @T @DERIVED 0 @T @T @DT @RT(12)tsODCStepPos @RT(0) @T @T @UNKNOWN 0 @F
@F @F
@T
@BEG_Attrib
3 @RT(0) @RT(0) @RT(0)
@END_Attrib
1 1 @F @F @F @F

@Var @RT(9)bNoAlarms @RT(0) @T @F @DT @RT(4)BOOL @RT(0) @T @T @BASIC 0 @F
@F @F
@T
@BEG_Attrib
3 @RT(0) @RT(52)TRUE: alarms of not fulfilled conditions are not set @RT(0)
@END_Attrib
1 1 @F @F @F @F

@Var @RT(18)bCheckConditionsOk @RT(0) @T @F @DT @RT(4)BOOL @RT(0) @T @T @BASIC 0 @F
@F @F
@T
@BEG_Attrib
3 @RT(0) @RT(0) @RT(0)
@END_Attrib
1 3 @F @F @F @F

@Var @RT(17)bStartConditionOk @RT(0) @T @F @DT @RT(4)BOOL @RT(0) @T @T @BASIC 0 @F
@F @F
@T
@BEG_Attrib
3 @RT(0) @RT(0) @RT(0)
@END_Attrib
1 3 @F @F @F @F

@Var @RT(20)bCheckConditionFound @RT(0) @T @F @DT @RT(4)BOOL @RT(0) @T @T @BASIC 0 @F
@F @F
@T
@BEG_Attrib
3 @RT(0) @RT(0) @RT(0)
@END_Attrib
1 3 @F @F @F @F

@Var @RT(1)i @RT(0) @T @F @DT @RT(4)DINT @RT(0) @T @T @BASIC 0 @F
@F @F
@T
@BEG_Attrib
3 @RT(0) @RT(0) @RT(0)
@END_Attrib
1 4 @F @F @F @F

@Var @RT(22)abODCCheckDependencies @RT(0) @T @T @DERIVED 0 @T @T @DT @RT(22)ABODCCheckDependencies @RT(0) @T @T @UNKNOWN 0 @F
@F @F
@T
@BEG_Attrib
3 @RT(0) @RT(0) @RT(0)
@END_Attrib
1 0 @F @F @F @F

@Var @RT(21)iStartConditionsNotOk @RT(0) @T @F @DT @RT(4)DINT @RT(0) @T @T @BASIC 0 @F
@F @F
@T
@BEG_Attrib
3 @RT(0) @RT(39)number of not fulfilled startconditions @RT(0)
@END_Attrib
1 3 @F @F @F @F

@Var @RT(21)iCheckConditionsNotOk @RT(0) @T @F @DT @RT(4)DINT @RT(0) @T @T @BASIC 0 @F
@F @F
@T
@BEG_Attrib
3 @RT(0) @RT(39)number of not fulfilled checkconditions @RT(0)
@END_Attrib
1 3 @F @F @F @F

@END_Dcl

@END_Export

@BEG_Export

@BEG_Algo
@ALGORITHM @RT(20)aStartSingleMovement @STRUCTURED_TEXT
@RT(0) @RT(0) @RT(0) @F @F
@END_Algo

@BEG_Dcl
@RT(16)DclTreeContainer
22
@Var @RT(8)DeviceId @RT(0) @T @T @DERIVED 0 @T @T @DT @RT(10)tsDeviceId @RT(0) @T @T @UNKNOWN 0 @F
@F @F
@T
@BEG_Attrib
3 @RT(0) @RT(0) @RT(0)
@END_Attrib
1 1 @F @F @F @F

@Var @RT(7)MoveDir @RT(0) @T @T @DERIVED 0 @T @T @DT @RT(10)tMoveIdent @RT(0) @T @T @UNKNOWN 0 @F
@F @F
@T
@BEG_Attrib
3 @RT(0) @RT(0) @RT(0)
@END_Attrib
1 1 @F @F @F @F

@Var @RT(6)MoveId @RT(0) @T @T @DERIVED 0 @T @T @DT @RT(10)tMoveIdent @RT(0) @T @T @UNKNOWN 0 @F
@F @F
@T
@BEG_Attrib
3 @RT(0) @RT(0) @RT(0)
@END_Attrib
1 1 @F @F @F @F

@Var @RT(16)IntermediateCond @RT(0) @T @F @DT @RT(4)DINT @RT(0) @T @T @BASIC 0 @F
@F @F
@T
@BEG_Attrib
3 @RT(0) @RT(0) @RT(0)
@END_Attrib
1 1 @F @F @F @F

@Var @RT(16)bNeedCheckSafety @RT(0) @T @F @DT @RT(4)BOOL @RT(0) @T @T @BASIC 0 @F
@F @F
@T
@BEG_Attrib
3 @RT(0) @RT(0) @RT(0)
@END_Attrib
1 1 @F @F @F @F

@Var @RT(7)StepPos @RT(0) @T @T @DERIVED 0 @T @T @DT @RT(12)tsODCStepPos @RT(0) @T @T @UNKNOWN 0 @F
@F @F
@T
@BEG_Attrib
3 @RT(0) @RT(0) @RT(0)
@END_Attrib
1 4 @F @F @F @F

@Var @RT(7)fbStart @RT(0) @T @T @DERIVED 0 @T @T @DT @RT(7)FBStart @RT(0) @T @T @UNKNOWN 0 @F
@F @F
@T
@BEG_Attrib
3 @RT(0) @RT(0) @RT(0)
@END_Attrib
1 0 @F @F @F @F

@Var @RT(27)abODCCheckDependenciesStart @RT(0) @T @T @DERIVED 0 @T @T @DT @RT(22)ABODCCheckDependencies @RT(0) @T @T @UNKNOWN 0 @F
@F @F
@T
@BEG_Attrib
3 @RT(0) @RT(0) @RT(0)
@END_Attrib
1 0 @F @F @F @F

@Var @RT(24)evCheckLocklistEventData @RT(0) @T @T @DERIVED 0 @T @T @DT @RT(20)tevCheckLocklistData @RT(0) @T @T @UNKNOWN 0 @F
@F @F
@T
@BEG_Attrib
3 @RT(0) @RT(0) @RT(0)
@END_Attrib
1 4 @F @F @F @F

@Var @RT(17)bStartConditionOk @RT(0) @T @F @DT @RT(4)BOOL @RT(0) @T @T @BASIC 0 @F
@F @F
@T
@BEG_Attrib
3 @RT(0) @RT(0) @RT(0)
@END_Attrib
1 0 @F @F @F @F

@Var @RT(18)bCheckConditionsOk @RT(0) @T @F @DT @RT(4)BOOL @RT(0) @T @T @BASIC 0 @F
@F @F
@T
@BEG_Attrib
3 @RT(0) @RT(0) @RT(0)
@END_Attrib
1 0 @F @F @F @F

@Var @RT(20)bCheckConditionFound @RT(0) @T @F @DT @RT(4)BOOL @RT(0) @T @T @BASIC 0 @F
@F @F
@T
@BEG_Attrib
3 @RT(0) @RT(0) @RT(0)
@END_Attrib
1 0 @F @F @F @F

@Var @RT(14)fbSetStepState @RT(0) @T @T @DERIVED 0 @T @T @DT @RT(14)FBSetStepState @RT(0) @T @T @UNKNOWN 0 @F
@F @F
@T
@BEG_Attrib
3 @RT(0) @RT(0) @RT(0)
@END_Attrib
1 0 @F @F @F @F

@Var @RT(17)bIgnoreConditions @RT(0) @T @F @DT @RT(4)BOOL @RT(0) @T @T @BASIC 0 @F
@F @F
@T
@BEG_Attrib
3 @RT(0) @RT(0) @RT(0)
@END_Attrib
1 0 @F @F @F @F

@Var @RT(15)bSearchMovement @RT(0) @T @F @DT @RT(4)BOOL @RT(0) @T @T @BASIC 0 @F
@F @F
@T
@BEG_Attrib
3 @RT(0) @RT(0) @RT(0)
@END_Attrib
1 0 @F @F @F @F

@Var @RT(14)bMovementFound @RT(0) @T @F @DT @RT(4)BOOL @RT(0) @T @T @BASIC 0 @F
@F @F
@T
@BEG_Attrib
3 @RT(0) @RT(0) @RT(0)
@END_Attrib
1 0 @F @F @F @F

@Var @RT(16)bMovementAllowed @RT(0) @T @F @DT @RT(4)BOOL @RT(0) @T @T @BASIC 0 @F
@F @F
@T
@BEG_Attrib
3 @RT(0) @RT(0) @RT(0)
@END_Attrib
1 0 @F @F @F @F

@Var @RT(10)TmpStepPos @RT(0) @T @T @DERIVED 0 @T @T @DT @RT(12)tsODCStepPos @RT(0) @T @T @UNKNOWN 0 @F
@F @F
@T
@BEG_Attrib
3 @RT(0) @RT(0) @RT(0)
@END_Attrib
1 0 @F @F @F @F

@Var @RT(14)iTmpAlarmCount @RT(0) @T @F @DT @RT(4)DINT @RT(0) @T @T @BASIC 0 @F
@F @F
@T
@BEG_Attrib
3 @RT(0) @RT(0) @RT(0)
@END_Attrib
1 0 @F @F @F @F

@Var @RT(19)StepPosLowestAlarms @RT(0) @T @T @DERIVED 0 @T @T @DT @RT(12)tsODCStepPos @RT(0) @T @T @UNKNOWN 0 @F
@F @F
@T
@BEG_Attrib
3 @RT(0) @RT(0) @RT(0)
@END_Attrib
1 0 @F @F @F @F

@Var @RT(11)iAlarmCount @RT(0) @T @F @DT @RT(4)DINT @RT(0) @T @T @BASIC 0 @F
@F @F
@T
@BEG_Attrib
3 @RT(0) @RT(0) @RT(0)
@END_Attrib
1 0 @F @F @F @F

@Var @RT(8)bStarted @RT(0) @T @F @DT @RT(4)BOOL @RT(0) @T @T @BASIC 0 @F
@F @F
@T
@BEG_Attrib
3 @RT(0) @RT(0) @RT(0)
@END_Attrib
1 3 @F @F @F @F

@END_Dcl

@END_Export

@BEG_Export

@BEG_Algo
@ALGORITHM @RT(22)aStartCombinedMovement @STRUCTURED_TEXT
@RT(0) @RT(0) @RT(0) @F @F
@END_Algo

@BEG_Dcl
@RT(16)DclTreeContainer
5
@Var @RT(8)DeviceId @RT(0) @T @T @DERIVED 0 @T @T @DT @RT(10)tsDeviceId @RT(0) @T @T @UNKNOWN 0 @F
@F @F
@T
@BEG_Attrib
3 @RT(0) @RT(0) @RT(0)
@END_Attrib
1 1 @F @F @F @F

@Var @RT(7)MoveDir @RT(0) @T @T @DERIVED 0 @T @T @DT @RT(10)tMoveIdent @RT(0) @T @T @UNKNOWN 0 @F
@F @F
@T
@BEG_Attrib
3 @RT(0) @RT(0) @RT(0)
@END_Attrib
1 1 @F @F @F @F

@Var @RT(6)MoveId @RT(0) @T @T @DERIVED 0 @T @T @DT @RT(10)tMoveIdent @RT(0) @T @T @UNKNOWN 0 @F
@F @F
@T
@BEG_Attrib
3 @RT(0) @RT(0) @RT(0)
@END_Attrib
1 1 @F @F @F @F

@Var @RT(8)StartPos @RT(0) @T @T @DERIVED 0 @T @T @DT @RT(12)tsODCStepPos @RT(0) @T @T @UNKNOWN 0 @F
@F @F
@T
@BEG_Attrib
3 @RT(0) @RT(0) @RT(0)
@END_Attrib
1 4 @F @F @F @F

@Var @RT(9)bNotFound @RT(0) @T @F @DT @RT(4)BOOL @RT(0) @T @T @BASIC 0 @F
@F @F
@T
@BEG_Attrib
3 @RT(0) @RT(0) @RT(0)
@END_Attrib
1 3 @F @F @F @F

@END_Dcl

@END_Export

@BEG_Export

@BEG_Algo
@EVENT_ALGORITHM @RT(15)evaStartRequest @STRUCTURED_TEXT
@RT(0) @RT(14)evStartRequest @RT(13)EV_Task_3(23) @F @F
@END_Algo

@BEG_Dcl
@RT(16)DclTreeContainer
6
@Var @RT(18)evStartRequestData @RT(0) @T @T @DERIVED 0 @T @T @DT @RT(19)tevStartRequestData @RT(0) @T @T @UNKNOWN 0 @F
@F @F
@T
@BEG_Attrib
3 @RT(0) @RT(0) @RT(0)
@END_Attrib
1 1 @F @F @F @F

@Var @RT(16)StartRequestData @RT(0) @T @T @DERIVED 0 @T @T @DT @RT(19)tevStartRequestData @RT(0) @T @T @UNKNOWN 0 @F
@F @F
@T
@BEG_Attrib
3 @RT(0) @RT(0) @RT(0)
@END_Attrib
1 0 @F @F @F @F

@Var @RT(12)bCheckSafety @RT(0) @T @F @DT @RT(4)BOOL @RT(0) @T @T @BASIC 0 @F
@F @F
@T
@BEG_Attrib
3 @RT(0) @RT(0) @RT(0)
@END_Attrib
1 0 @F @F @F @F

@Var @RT(7)iSafety @RT(0) @T @F @DT @RT(4)DINT @RT(0) @T @T @BASIC 0 @F
@F @F
@T
@BEG_Attrib
3 @RT(0) @RT(0) @RT(0)
@END_Attrib
1 0 @F @F @F @F

@Var @RT(9)bCombined @RT(0) @T @F @DT @RT(4)BOOL @RT(0) @T @T @BASIC 0 @F
@F @F
@T
@BEG_Attrib
3 @RT(0) @RT(0) @RT(0)
@END_Attrib
1 0 @F @F @F @F

@Var @RT(1)i @RT(0) @T @F @DT @RT(4)DINT @RT(0) @T @T @BASIC 0 @F
@F @F
@T
@BEG_Attrib
3 @RT(0) @RT(0) @RT(0)
@END_Attrib
1 4 @F @F @F @F

@END_Dcl

@END_Export

@BEG_Export

@BEG_Algo
@EVENT_ALGORITHM @RT(14)evaStopRequest @STRUCTURED_TEXT
@RT(0) @RT(13)evStopRequest @RT(9)EV_Task_3 @F @F
@END_Algo

@BEG_Dcl
@RT(16)DclTreeContainer
2
@Var @RT(17)evStopRequestData @RT(0) @T @T @DERIVED 0 @T @T @DT @RT(18)tevStopRequestData @RT(0) @T @T @UNKNOWN 0 @F
@F @F
@T
@BEG_Attrib
3 @RT(0) @RT(0) @RT(0)
@END_Attrib
1 1 @F @F @F @F

@Var @RT(6)fbStop @RT(0) @T @T @DERIVED 0 @T @T @DT @RT(6)FBStop @RT(0) @T @T @UNKNOWN 0 @F
@F @F
@T
@BEG_Attrib
3 @RT(0) @RT(0) @RT(0)
@END_Attrib
1 0 @F @F @F @F

@END_Dcl

@END_Export

@BEG_Export

@BEG_Algo
@ALGORITHM @RT(19)aDecreaseLineNumber @STRUCTURED_TEXT
@RT(0) @RT(0) @RT(0) @F @F
@END_Algo

@BEG_Dcl
@RT(16)DclTreeContainer
7
@Var @RT(8)DeviceId @RT(0) @T @T @DERIVED 0 @T @T @DT @RT(10)tsDeviceId @RT(0) @T @T @UNKNOWN 0 @F
@F @F
@T
@BEG_Attrib
3 @RT(0) @RT(0) @RT(0)
@END_Attrib
1 1 @F @F @F @F

@Var @RT(6)MoveId @RT(0) @T @T @DERIVED 0 @T @T @DT @RT(10)tMoveIdent @RT(0) @T @T @UNKNOWN 0 @F
@F @F
@T
@BEG_Attrib
3 @RT(0) @RT(0) @RT(0)
@END_Attrib
1 1 @F @F @F @F

@Var @RT(7)MoveDir @RT(0) @T @T @DERIVED 0 @T @T @DT @RT(10)tMoveIdent @RT(0) @T @T @UNKNOWN 0 @F
@F @F
@T
@BEG_Attrib
3 @RT(0) @RT(0) @RT(0)
@END_Attrib
1 1 @F @F @F @F

@Var @RT(17)fbCheckPosReached @RT(0) @T @T @DERIVED 0 @T @T @DT @RT(17)FBCheckPosReached @RT(0) @T @T @UNKNOWN 0 @F
@F @F
@T
@BEG_Attrib
3 @RT(0) @RT(0) @RT(0)
@END_Attrib
1 0 @F @F @F @F

@Var @RT(10)iTmpColumn @RT(0) @T @F @DT @RT(4)DINT @RT(0) @T @T @BASIC 0 @F
@F @F
@T
@BEG_Attrib
3 @RT(0) @RT(0) @RT(0)
@END_Attrib
1 4 @F @F @F @F

@Var @RT(1)i @RT(0) @T @F @DT @RT(4)DINT @RT(0) @T @T @BASIC 0 @F
@F @F
@T
@BEG_Attrib
3 @RT(0) @RT(0) @RT(0)
@END_Attrib
1 4 @F @F @F @F

@Var @RT(5)dummy @RT(0) @T @F @DT @RT(4)DINT @RT(0) @T @T @BASIC 0 @F
@F @F
@T
@BEG_Attrib
3 @RT(0) @RT(0) @RT(0)
@END_Attrib
1 0 @F @F @F @F

@END_Dcl

@END_Export

@BEG_Export

@BEG_Algo
@EVENT_ALGORITHM @RT(17)evaStartedStopped @STRUCTURED_TEXT
@RT(0) @RT(16)evStartedStopped @RT(9)EV_Task_3 @F @F
@END_Algo

@BEG_Dcl
@RT(16)DclTreeContainer
8
@Var @RT(20)evStartedStoppedData @RT(0) @T @T @DERIVED 0 @T @T @DT @RT(21)tevStartedStoppedData @RT(0) @T @T @UNKNOWN 0 @F
@F @F
@T
@BEG_Attrib
3 @RT(0) @RT(0) @RT(0)
@END_Attrib
1 1 @F @F @F @F

@Var @RT(11)tmpMovement @RT(0) @T @T @DERIVED 0 @T @T @DT @RT(28)tsStartedMoveInfoODCExtended @RT(0) @T @T @UNKNOWN 0 @F
@F @F
@T
@BEG_Attrib
3 @RT(0) @RT(0) @RT(0)
@END_Attrib
1 4 @F @F @F @F

@Var @RT(1)i @RT(0) @T @F @DT @RT(4)DINT @RT(0) @T @T @BASIC 0 @F
@F @F
@T
@BEG_Attrib
3 @RT(0) @RT(0) @RT(0)
@END_Attrib
1 4 @F @F @F @F

@Var @RT(6)bFound @RT(0) @T @F @DT @RT(4)BOOL @RT(0) @T @T @BASIC 0 @F
@F @F
@T
@BEG_Attrib
3 @RT(0) @RT(0) @RT(0)
@END_Attrib
1 0 @F @F @F @F

@Var @RT(7)stepPos @RT(0) @T @T @DERIVED 0 @T @T @DT @RT(12)tsODCStepPos @RT(0) @T @T @UNKNOWN 0 @F
@F @F
@T
@BEG_Attrib
3 @RT(0) @RT(0) @RT(0)
@END_Attrib
1 4 @F @F @F @F

@Var @RT(3)idx @RT(0) @T @F @DT @RT(4)DINT @RT(0) @T @T @BASIC 0 @F
@F @F
@T
@BEG_Attrib
3 @RT(0) @RT(0) @RT(0)
@END_Attrib
1 4 @F @F @F @F

@Var @RT(14)fbSetStepState @RT(0) @T @T @DERIVED 0 @T @T @DT @RT(14)FBSetStepState @RT(0) @T @T @UNKNOWN 0 @F
@F @F
@T
@BEG_Attrib
3 @RT(0) @RT(0) @RT(0)
@END_Attrib
1 0 @F @F @F @F

@Var @RT(16)bCorrectInstance @RT(0) @T @F @DT @RT(4)BOOL @RT(0) @T @T @BASIC 0 @F
@F @F
@T
@BEG_Attrib
3 @RT(0) @RT(0) @RT(0)
@END_Attrib
1 0 @F @F @F @F

@END_Dcl

@END_Export

@BEG_Export

@BEG_Algo
@POSTUPDATE_ALGORITHM @RT(17)pStartedMovements @STRUCTURED_TEXT
@RT(0) @RT(43)sv_StartedManualMovements.iStartedMovements @RT(9)PU_Task_3 @F @F
@END_Algo

@BEG_Dcl
@RT(16)DclTreeContainer
0
@END_Dcl

@END_Export

@BEG_Export

@BEG_Algo
@PROCESS_ALGORITHM @RT(22)paCyclicConditionCheck @STRUCTURED_TEXT
@RT(0) @RT(0) @RT(10)TaskAnalog @F @F
@END_Algo

@BEG_Dcl
@RT(16)DclTreeContainer
3
@Var @RT(1)i @RT(0) @T @F @DT @RT(4)DINT @RT(0) @T @T @BASIC 0 @F
@F @F
@T
@BEG_Attrib
3 @RT(0) @RT(0) @RT(0)
@END_Attrib
1 4 @F @F @F @F

@Var @RT(28)abODCCheckDependenciesCyclic @RT(0) @T @T @DERIVED 0 @T @T @DT @RT(22)ABODCCheckDependencies @RT(0) @T @T @UNKNOWN 0 @F
@F @F
@T
@BEG_Attrib
3 @RT(0) @RT(83)must be a separate block since it is accessed from different tasks at the same time @RT(0)
@END_Attrib
1 0 @F @F @F @F

@Var @RT(10)TmpStepPos @RT(0) @T @T @DERIVED 0 @T @T @DT @RT(12)tsODCStepPos @RT(0) @T @T @UNKNOWN 0 @F
@F @F
@T
@BEG_Attrib
3 @RT(0) @RT(0) @RT(0)
@END_Attrib
1 0 @F @F @F @F

@END_Dcl

@END_Export

@BEG_Export

@BEG_Algo
@ALGORITHM @RT(13)aRunAutoCycle @SEQUENTIAL_FLOW_CHART
@RT(0) @RT(0) @RT(0) @F @F
@END_Algo

@BEG_Dcl
@RT(16)DclTreeContainer
17
@Var @RT(10)bStopCycle @RT(0) @T @F @DT @RT(4)BOOL @RT(0) @T @T @BASIC 0 @F
@F @F
@T
@BEG_Attrib
3 @RT(0) @RT(22)stop cycle immediately @RT(0)
@END_Attrib
1 1 @F @F @F @F

@Var @RT(15)bStopAfterCycle @RT(0) @T @F @DT @RT(4)BOOL @RT(0) @T @T @BASIC 0 @F
@F @F
@T
@BEG_Attrib
3 @RT(0) @RT(32)finish the actual cycle and stop @RT(0)
@END_Attrib
1 1 @F @F @F @F

@Var @RT(6)bReady @RT(0) @T @F @DT @RT(4)BOOL @RT(0) @T @T @BASIC 0 @F
@F @F
@T
@BEG_Attrib
3 @RT(0) @RT(0) @RT(0)
@END_Attrib
1 3 @F @F @F @F

@Var @RT(9)bCanStart @RT(0) @T @F @DT @RT(4)BOOL @RT(0) @T @T @BASIC 0 @F
@F @F
@T
@BEG_Attrib
3 @RT(0) @RT(75)got the cycle start signal-> cycle can start if sequence recalc is finished @RT(0)
@END_Attrib
1 0 @F @F @F @F

@Var @RT(16)abWaitCycleStart @RT(0) @T @T @DERIVED 0 @T @T @DT @RT(16)ABWaitCycleStart @RT(0) @T @T @UNKNOWN 0 @F
@F @F
@T
@BEG_Attrib
3 @RT(0) @RT(0) @RT(0)
@END_Attrib
1 0 @F @F @F @F

@Var @RT(7)fbStart @RT(0) @T @T @DERIVED 0 @T @T @DT @RT(7)FBStart @RT(0) @T @T @UNKNOWN 0 @F
@F @F
@T
@BEG_Attrib
3 @RT(0) @RT(0) @RT(0)
@END_Attrib
1 0 @F @F @F @F

@Var @RT(14)bDelayExceeded @RT(0) @T @F @DT @RT(4)BOOL @RT(0) @T @T @BASIC 0 @F
@F @F
@T
@BEG_Attrib
3 @RT(0) @RT(0) @RT(0)
@END_Attrib
1 0 @F @F @F @F

@Var @RT(18)bEjectorBwdStarted @RT(0) @T @F @DT @RT(4)BOOL @RT(0) @T @T @BASIC 0 @F
@F @F
@T
@BEG_Attrib
3 @RT(0) @RT(0) @RT(0)
@END_Attrib
1 0 @F @F @F @F

@Var @RT(15)DeviceIdEjector @RT(0) @T @T @DERIVED 0 @T @T @DT @RT(10)tsDeviceId @RT(0) @T @T @UNKNOWN 0 @F
@F @F
@T
@BEG_Attrib
3 @RT(33)(CompId:=cCompEjector,IndexId:=1) @RT(0) @RT(0)
@END_Attrib
1 0 @F @F @F @F

@Var @RT(9)bInitDone @RT(0) @T @F @DT @RT(4)BOOL @RT(0) @T @T @BASIC 0 @F
@F @F
@T
@BEG_Attrib
3 @RT(0) @RT(0) @RT(0)
@END_Attrib
1 0 @F @F @F @F

@Var @RT(12)pbEjectorBwd @RT(0) @T @T @REFTO 0 @T @DT @RT(4)BOOL @RT(0) @T @T @BASIC 0 @F
@F @F
@T
@BEG_Attrib
3 @RT(0) @RT(0) @RT(0)
@END_Attrib
1 0 @F @F @F @F

@Var @RT(21)pbEjectorBwdActivated @RT(0) @T @T @REFTO 0 @T @DT @RT(4)BOOL @RT(0) @T @T @BASIC 0 @F
@F @F
@T
@BEG_Attrib
3 @RT(0) @RT(0) @RT(0)
@END_Attrib
1 0 @F @F @F @F

@Var @RT(14)pbEjectorReady @RT(0) @T @T @REFTO 0 @T @DT @RT(4)BOOL @RT(0) @T @T @BASIC 0 @F
@F @F
@T
@BEG_Attrib
3 @RT(0) @RT(0) @RT(0)
@END_Attrib
1 0 @F @F @F @F

@Var @RT(17)iMoveNrEjectorBwd @RT(0) @T @F @DT @RT(4)DINT @RT(0) @T @T @BASIC 0 @F
@F @F
@T
@BEG_Attrib
3 @RT(0) @RT(0) @RT(0)
@END_Attrib
1 0 @F @F @F @F

@Var @RT(13)bColumnActive @RT(0) @T @F @DT @RT(4)BOOL @RT(0) @T @T @BASIC 0 @F
@F @F
@T
@BEG_Attrib
3 @RT(0) @RT(0) @RT(0)
@END_Attrib
1 0 @F @F @F @F

@Var @RT(9)bDoRecalc @RT(0) @T @F @DT @RT(4)BOOL @RT(0) @T @T @BASIC 0 @F
@F @F
@T
@BEG_Attrib
3 @RT(0) @RT(0) @RT(0)
@END_Attrib
1 0 @F @F @F @F

@Var @RT(20)bMovesBeforeAutoLoop @RT(0) @T @F @DT @RT(4)BOOL @RT(0) @T @T @BASIC 0 @F
@F @F
@T
@BEG_Attrib
3 @RT(0) @RT(0) @RT(0)
@END_Attrib
1 0 @F @F @F @F

@END_Dcl

@END_Export

@BEG_Export

@BEG_Algo
@PROCESS_ALGORITHM @RT(23)paRunAutomaticMovements @STRUCTURED_TEXT
@RT(0) @RT(0) @RT(13)TaskSequencer @F @F
@END_Algo

@BEG_Dcl
@RT(16)DclTreeContainer
0
@END_Dcl

@END_Export

@BEG_Export

@BEG_Algo
@POSTUPDATE_ALGORITHM @RT(9)pInitDone @STRUCTURED_TEXT
@RT(0) @RT(12)sv_bInitDone @RT(9)PU_Task_3 @F @F
@END_Algo

@BEG_Dcl
@RT(16)DclTreeContainer
0
@END_Dcl

@END_Export

@BEG_Export

@BEG_Algo
@PROCESS_ALGORITHM @RT(6)paInit @STRUCTURED_TEXT
@RT(0) @RT(0) @RT(7)TaskMid @T @F
@END_Algo

@BEG_Dcl
@RT(16)DclTreeContainer
1
@Var @RT(8)swoState @RT(0) @T @T @DERIVED 0 @T @T @DT @RT(11)KSWO_Status @RT(0) @T @T @UNKNOWN 0 @F
@F @F
@T
@BEG_Attrib
3 @RT(0) @RT(0) @RT(0)
@END_Attrib
1 0 @F @F @F @F

@END_Dcl

@END_Export

@BEG_Export

@BEG_Algo
@POSTUPDATE_ALGORITHM @RT(14)pOpmodeChanged @STRUCTURED_TEXT
@RT(0) @RT(16)sv_OperationMode @RT(9)PU_Task_7 @F @F
@END_Algo

@BEG_Dcl
@RT(16)DclTreeContainer
0
@END_Dcl

@END_Export

@BEG_Export

@BEG_Algo
@EVENT_ALGORITHM @RT(21)evaFinishCycleAndStop @STRUCTURED_TEXT
@RT(0) @RT(25)evAlarmFinishCycleAndStop @RT(9)EV_Task_3 @F @F
@END_Algo

@BEG_Dcl
@RT(16)DclTreeContainer
1
@Var @RT(24)evFinishCycleAndStopData @RT(0) @T @T @DERIVED 0 @T @T @DT @RT(16)ALARM_EVENT_DATA @RT(0) @T @T @UNKNOWN 0 @F
@F @F
@T
@BEG_Attrib
3 @RT(0) @RT(0) @RT(0)
@END_Attrib
1 1 @F @F @F @F

@END_Dcl

@END_Export

@BEG_Export

@BEG_Algo
@POSTUPDATE_ALGORITHM @RT(10)pDataState @STRUCTURED_TEXT
@RT(0) @RT(12)sv_DataState @RT(12)PU_Task_3(1) @F @F
@END_Algo

@BEG_Dcl
@RT(16)DclTreeContainer
1
@Var @RT(9)PrevState @RT(0) @T @T @DERIVED 0 @T @T @DT @RT(11)tnDataState @RT(0) @T @T @UNKNOWN 0 @F
@F @F
@T
@BEG_Attrib
3 @RT(0) @RT(0) @RT(0)
@END_Attrib
1 0 @F @F @F @F

@END_Dcl

@END_Export

@BEG_Export

@BEG_Algo
@POSTUPDATE_ALGORITHM @RT(24)pDescriptionFilesChanged @STRUCTURED_TEXT
@RT(0) @RT(19)sv_bODCFilesChanged @RT(9)PU_Task_3 @F @F
@END_Algo

@BEG_Dcl
@RT(16)DclTreeContainer
0
@END_Dcl

@END_Export

@BEG_Export

@BEG_Algo
@POSTUPDATE_ALGORITHM @RT(22)pNewSequenceFromEditor @STRUCTURED_TEXT
@RT(0) @RT(17)sv_iActiveEditors @RT(9)PU_Task_3 @F @F
@END_Algo

@BEG_Dcl
@RT(16)DclTreeContainer
1
@Var @RT(12)fbLockUnlock @RT(0) @T @T @DERIVED 0 @T @T @DT @RT(12)FBLockUnlock @RT(0) @T @T @UNKNOWN 0 @F
@F @F
@T
@BEG_Attrib
3 @RT(98)(DeviceId:=(CompId:=cCompOperationMode,IndexId:=1),MoveDir:=cModeAutomatic,MoveId:=cModeAutomatic) @RT(0) @RT(0)
@END_Attrib
1 0 @F @F @F @F

@END_Dcl

@END_Export

@BEG_Export

@BEG_Algo
@POSTUPDATE_ALGORITHM @RT(22)aRestoreSequenceBackup @STRUCTURED_TEXT
@RT(0) @RT(21)sv_iSequenceToRestore @RT(9)EV_Task_7 @F @F
@END_Algo

@BEG_Dcl
@RT(16)DclTreeContainer
0
@END_Dcl

@END_Export
